LIN {X 0,Y 624.89,Z 336.382,A -85,B 0,C 180,E1 22685.786,E2 22685.786} C_VEL
LIN {X 0,Y 624.904,Z 336.388,A -85,B 0,C 180,E1 22682.935,E2 22682.935} C_VEL
LIN {X 0,Y 624.889,Z 336.39,A -85,B 0,C 180,E1 22679.725,E2 22679.725} C_VEL
LIN {X 0,Y 624.882,Z 336.387,A -85,B 0,C 180,E1 22676.973,E2 22676.973} C_VEL
LIN {X 0,Y 624.896,Z 336.39,A -85,B 0,C 180,E1 22673.753,E2 22673.753} C_VEL
LIN {X 0,Y 624.864,Z 336.382,A -85,B 0,C 180,E1 22671.071,E2 22671.071} C_VEL
LIN {X 0,Y 624.941,Z 336.367,A -85,B 0,C 180,E1 22668.089,E2 22668.089} C_VEL
LIN {X 0,Y 624.856,Z 336.372,A -85,B 0,C 180,E1 22665.129,E2 22665.129} C_VEL
LIN {X 0,Y 624.887,Z 336.388,A -85,B 0,C 180,E1 22662.397,E2 22662.397} C_VEL
LIN {X 0,Y 624.855,Z 336.37,A -85,B 0,C 180,E1 22659.192,E2 22659.192} C_VEL
LIN {X 0,Y 624.852,Z 336.393,A -85,B 0,C 180,E1 22656.618,E2 22656.618} C_VEL
LIN {X 0,Y 624.897,Z 336.367,A -85,B 0,C 180,E1 22653.485,E2 22653.485} C_VEL
LIN {X 0,Y 624.852,Z 336.389,A -85,B 0,C 180,E1 22650.681,E2 22650.681} C_VEL
LIN {X 0,Y 624.926,Z 336.387,A -85,B 0,C 180,E1 22647.805,E2 22647.805} C_VEL
LIN {X 0,Y 624.867,Z 336.396,A -85,B 0,C 180,E1 22644.826,E2 22644.826} C_VEL
LIN {X 0,Y 624.909,Z 336.51,A -85,B 0,C 180,E1 22644.021,E2 22644.021} C_VEL
LIN {X 0,Y 626.185,Z 339.775,A -85,B 0,C 180,E1 22643.558,E2 22643.558} C_VEL
LIN {X 0,Y 627.184,Z 341.437,A -85,B 0,C 180,E1 22643.284,E2 22643.284} C_VEL
LIN {X 0,Y 631.826,Z 350.571,A -85,B 0,C 180,E1 22641.946,E2 22641.946} C_VEL
LIN {X 0,Y 646.023,Z 370.4,A -85,B 0,C 180,E1 22640.049,E2 22640.049} C_VEL
LIN {X 0,Y 658.613,Z 388.736,A -85,B 0,C 180,E1 22638.466,E2 22638.466} C_VEL
LIN {X 0,Y 661.685,Z 393.59,A -85,B 0,C 180,E1 22638.09,E2 22638.09} C_VEL
LIN {X 0,Y 657.538,Z 599.762,A -85,B 0,C 180,E1 22635.27,E2 22635.27} C_VEL
LIN {X 0,Y 653.324,Z 821.102,A -85,B 0,C 180,E1 22632.317,E2 22632.317} C_VEL
LIN {X 0,Y 652.435,Z 844.522,A -85,B 0,C 180,E1 22631.931,E2 22631.931} C_VEL
LIN {X 0,Y 651.298,Z 867.206,A -85,B 0,C 180,E1 22631.437,E2 22631.437} C_VEL
LIN {X 0,Y 649.719,Z 893.305,A -85,B 0,C 180,E1 22630.717,E2 22630.717} C_VEL
LIN {X 0,Y 647.798,Z 918.713,A -85,B 0,C 180,E1 22629.833,E2 22629.833} C_VEL
LIN {X 0,Y 645.976,Z 940.579,A -85,B 0,C 180,E1 22628.935,E2 22628.935} C_VEL
LIN {X 0,Y 644.088,Z 961.696,A -85,B 0,C 180,E1 22627.934,E2 22627.934} C_VEL
LIN {X 0,Y 641.747,Z 986.505,A -85,B 0,C 180,E1 22626.581,E2 22626.581} C_VEL
LIN {X 0,Y 639.476,Z 1008.583,A -85,B 0,C 180,E1 22625.183,E2 22625.183} C_VEL
LIN {X 0,Y 637.567,Z 1026.895,A -85,B 0,C 180,E1 22623.885,E2 22623.885} C_VEL
LIN {X 0,Y 635.699,Z 1044.654,A -85,B 0,C 180,E1 22622.489,E2 22622.489} C_VEL
LIN {X 0,Y 633.544,Z 1065.5,A -85,B 0,C 180,E1 22620.667,E2 22620.667} C_VEL
LIN {X 0,Y 631.512,Z 1085.194,A -85,B 0,C 180,E1 22618.697,E2 22618.697} C_VEL
LIN {X 0,Y 630.037,Z 1100.529,A -85,B 0,C 180,E1 22616.994,E2 22616.994} C_VEL
LIN {X 0,Y 628.438,Z 1118.006,A -85,B 0,C 180,E1 22614.837,E2 22614.837} C_VEL
LIN {X 0,Y 627.119,Z 1133.826,A -85,B 0,C 180,E1 22612.597,E2 22612.597} C_VEL
LIN {X 0,Y 626.192,Z 1146.58,A -85,B 0,C 180,E1 22610.566,E2 22610.566} C_VEL
LIN {X 0,Y 625.357,Z 1159.888,A -85,B 0,C 180,E1 22608.167,E2 22608.167} C_VEL
LIN {X 0,Y 624.744,Z 1171.078,A -85,B 0,C 180,E1 22605.788,E2 22605.788} C_VEL
LIN {X 0,Y 624.417,Z 1179.159,A -85,B 0,C 180,E1 22603.804,E2 22603.804} C_VEL
LIN {X 0,Y 624.174,Z 1186.705,A -85,B 0,C 180,E1 22601.645,E2 22601.645} C_VEL
LIN {X 0,Y 624.015,Z 1193.594,A -85,B 0,C 180,E1 22599.221,E2 22599.221} C_VEL
LIN {X 0,Y 623.939,Z 1198.918,A -85,B 0,C 180,E1 22596.718,E2 22596.718} C_VEL
LIN {X 0,Y 623.915,Z 1202.24,A -85,B 0,C 180,E1 22594.504,E2 22594.504} C_VEL
LIN {X 0,Y 623.912,Z 1204.382,A -85,B 0,C 180,E1 22592.113,E2 22592.113} C_VEL
LIN {X 0,Y 623.892,Z 1204.894,A -85,B 0,C 180,E1 22589.541,E2 22589.541} C_VEL
LIN {X 0,Y 623.911,Z 1204.004,A -85,B 0,C 180,E1 22587.337,E2 22587.337} C_VEL
LIN {X 0,Y 623.923,Z 1201.672,A -85,B 0,C 180,E1 22585.036,E2 22585.036} C_VEL
LIN {X 0,Y 623.958,Z 1197.543,A -85,B 0,C 180,E1 22582.542,E2 22582.542} C_VEL
LIN {X 0,Y 624.046,Z 1191.873,A -85,B 0,C 180,E1 22580.129,E2 22580.129} C_VEL
LIN {X 0,Y 624.21,Z 1184.888,A -85,B 0,C 180,E1 22577.794,E2 22577.794} C_VEL
LIN {X 0,Y 624.578,Z 1175.442,A -85,B 0,C 180,E1 22575.229,E2 22575.229} C_VEL
LIN {X 0,Y 625.05,Z 1164.999,A -85,B 0,C 180,E1 22572.882,E2 22572.882} C_VEL
LIN {X 0,Y 625.664,Z 1154.466,A -85,B 0,C 180,E1 22570.821,E2 22570.821} C_VEL
LIN {X 0,Y 626.612,Z 1140.788,A -85,B 0,C 180,E1 22568.469,E2 22568.469} C_VEL
LIN {X 0,Y 627.822,Z 1125.095,A -85,B 0,C 180,E1 22566.139,E2 22566.139} C_VEL
LIN {X 0,Y 629.06,Z 1111.083,A -85,B 0,C 180,E1 22564.283,E2 22564.283} C_VEL
LIN {X 0,Y 630.77,Z 1092.862,A -85,B 0,C 180,E1 22562.12,E2 22562.12} C_VEL
LIN {X 0,Y 632.664,Z 1073.813,A -85,B 0,C 180,E1 22560.144,E2 22560.144} C_VEL
LIN {X 0,Y 634.359,Z 1057.391,A -85,B 0,C 180,E1 22558.606,E2 22558.606} C_VEL
LIN {X 0,Y 636.32,Z 1038.638,A -85,B 0,C 180,E1 22557.017,E2 22557.017} C_VEL
LIN {X 0,Y 638.858,Z 1014.535,A -85,B 0,C 180,E1 22555.222,E2 22555.222} C_VEL
LIN {X 0,Y 640.898,Z 994.594,A -85,B 0,C 180,E1 22553.916,E2 22553.916} C_VEL
LIN {X 0,Y 642.856,Z 974.946,A -85,B 0,C 180,E1 22552.769,E2 22552.769} C_VEL
LIN {X 0,Y 645.084,Z 951.666,A -85,B 0,C 180,E1 22551.571,E2 22551.571} C_VEL
LIN {X 0,Y 647.218,Z 926.44,A -85,B 0,C 180,E1 22550.47,E2 22550.47} C_VEL
LIN {X 0,Y 648.844,Z 904.861,A -85,B 0,C 180,E1 22549.668,E2 22549.668} C_VEL
LIN {X 0,Y 650.326,Z 883.219,A -85,B 0,C 180,E1 22548.988,E2 22548.988} C_VEL
LIN {X 0,Y 651.688,Z 860.13,A -85,B 0,C 180,E1 22548.394,E2 22548.394} C_VEL
LIN {X 0,Y 652.995,Z 831.823,A -85,B 0,C 180,E1 22547.842,E2 22547.842} C_VEL
LIN {X 0,Y 654.187,Z 777.579,A -85,B 0,C 180,E1 22547.102,E2 22547.102} C_VEL
LIN {X 0,Y 658.412,Z 555.546,A -85,B 0,C 180,E1 22544.133,E2 22544.133} C_VEL
LIN {X 0,Y 661.622,Z 393.144,A -85,B 0,C 180,E1 22541.897,E2 22541.897} C_VEL
LIN {X 0,Y 647.935,Z 373.153,A -85,B 0,C 180,E1 22540.199,E2 22540.199} C_VEL
LIN {X 0,Y 638.133,Z 359.287,A -85,B 0,C 180,E1 22538.898,E2 22538.898} C_VEL
LIN {X 0,Y 631.374,Z 349.693,A -85,B 0,C 180,E1 22537.913,E2 22537.913} C_VEL
LIN {X 0,Y 627.309,Z 341.424,A -85,B 0,C 180,E1 22536.594,E2 22536.594} C_VEL
LIN {X 0,Y 625.187,Z 337.75,A -85,B 0,C 180,E1 22535.942,E2 22535.942} C_VEL
LIN {X 0,Y 624.876,Z 336.385,A -85,B 0,C 180,E1 22535.736,E2 22535.736} C_VEL
LIN {X 0,Y 624.878,Z 336.391,A -85,B 0,C 180,E1 22532.96,E2 22532.96} C_VEL
LIN {X 0,Y 624.872,Z 336.375,A -85,B 0,C 180,E1 22529.633,E2 22529.633} C_VEL
LIN {X 0,Y 624.86,Z 336.37,A -85,B 0,C 180,E1 22526.966,E2 22526.966} C_VEL
LIN {X 0,Y 624.91,Z 336.391,A -85,B 0,C 180,E1 22523.88,E2 22523.88} C_VEL
LIN {X 0,Y 624.848,Z 336.368,A -85,B 0,C 180,E1 22521.103,E2 22521.103} C_VEL
LIN {X 0,Y 624.899,Z 336.383,A -85,B 0,C 180,E1 22518.277,E2 22518.277} C_VEL
LIN {X 0,Y 624.853,Z 336.384,A -85,B 0,C 180,E1 22515.215,E2 22515.215} C_VEL
LIN {X 0,Y 624.854,Z 336.38,A -85,B 0,C 180,E1 22512.57,E2 22512.57} C_VEL
LIN {X 0,Y 624.884,Z 336.388,A -85,B 0,C 180,E1 22509.393,E2 22509.393} C_VEL
LIN {X 0,Y 624.85,Z 336.372,A -85,B 0,C 180,E1 22506.708,E2 22506.708} C_VEL
LIN {X 0,Y 624.929,Z 336.381,A -85,B 0,C 180,E1 22503.761,E2 22503.761} C_VEL
LIN {X 0,Y 624.857,Z 336.362,A -85,B 0,C 180,E1 22500.733,E2 22500.733} C_VEL
LIN {X 0,Y 624.88,Z 336.388,A -85,B 0,C 180,E1 22498.074,E2 22498.074} C_VEL
LIN {X 0,Y 624.877,Z 336.356,A -85,B 0,C 180,E1 22494.859,E2 22494.859} C_VEL
LIN {X 0,Y 624.873,Z 336.392,A -85,B 0,C 180,E1 22492.183,E2 22492.183} C_VEL
LIN {X 0,Y 624.929,Z 336.355,A -85,B 0,C 180,E1 22489.117,E2 22489.117} C_VEL
LIN {X 0,Y 624.874,Z 336.39,A -85,B 0,C 180,E1 22486.206,E2 22486.206} C_VEL
LIN {X 0,Y 624.946,Z 336.36,A -85,B 0,C 180,E1 22483.262,E2 22483.262} C_VEL
LIN {X 0,Y 624.878,Z 336.366,A -85,B 0,C 180,E1 22480.196,E2 22480.196} C_VEL
LIN {X 0,Y 624.932,Z 336.391,A -85,B 0,C 180,E1 22477.319,E2 22477.319} C_VEL
LIN {X 0,Y 624.889,Z 336.375,A -85,B 0,C 180,E1 22474.2,E2 22474.2} C_VEL
LIN {X 0,Y 624.91,Z 336.39,A -85,B 0,C 180,E1 22471.418,E2 22471.418} C_VEL
LIN {X 0,Y 624.933,Z 336.553,A -85,B 0,C 180,E1 22469.363,E2 22469.363} C_VEL
LIN {X 0,Y 626.26,Z 339.858,A -85,B 0,C 180,E1 22468.844,E2 22468.844} C_VEL
LIN {X 0,Y 627.438,Z 341.862,A -85,B 0,C 180,E1 22468.499,E2 22468.499} C_VEL
LIN {X 0,Y 630.498,Z 346.011,A -85,B 0,C 180,E1 22468.043,E2 22468.043} C_VEL
LIN {X 0,Y 638.814,Z 357.205,A -85,B 0,C 180,E1 22466.862,E2 22466.862} C_VEL
LIN {X 0,Y 649.952,Z 372.837,A -85,B 0,C 180,E1 22465.398,E2 22465.398} C_VEL
LIN {X 0,Y 661.396,Z 389.816,A -85,B 0,C 180,E1 22463.978,E2 22463.978} C_VEL
LIN {X 0,Y 661.577,Z 391.519,A -85,B 0,C 180,E1 22463.934,E2 22463.934} C_VEL
LIN {X 0,Y 659.206,Z 504.502,A -85,B 0,C 180,E1 22462.383,E2 22462.383} C_VEL
LIN {X 0,Y 658.369,Z 512.206,A -85,B 0,C 180,E1 22462.34,E2 22462.34} C_VEL
LIN {X 0,Y 653.608,Z 532.876,A -85,B 0,C 180,E1 22462.456,E2 22462.456} C_VEL
LIN {X 0,Y 652.955,Z 539.485,A -85,B 0,C 180,E1 22462.413,E2 22462.413} C_VEL
LIN {X 0,Y 648.476,Z 760.283,A -85,B 0,C 180,E1 22459.432,E2 22459.432} C_VEL
LIN {X 0,Y 647.121,Z 819.424,A -85,B 0,C 180,E1 22458.626,E2 22458.626} C_VEL
LIN {X 0,Y 645.939,Z 846.309,A -85,B 0,C 180,E1 22458.126,E2 22458.126} C_VEL
LIN {X 0,Y 644.286,Z 872.533,A -85,B 0,C 180,E1 22457.46,E2 22457.46} C_VEL
LIN {X 0,Y 642.784,Z 893.338,A -85,B 0,C 180,E1 22456.807,E2 22456.807} C_VEL
LIN {X 0,Y 641.188,Z 912.912,A -85,B 0,C 180,E1 22456.091,E2 22456.091} C_VEL
LIN {X 0,Y 639.312,Z 933.875,A -85,B 0,C 180,E1 22455.203,E2 22455.203} C_VEL
LIN {X 0,Y 636.999,Z 958.427,A -85,B 0,C 180,E1 22453.999,E2 22453.999} C_VEL
LIN {X 0,Y 634.522,Z 981.775,A -85,B 0,C 180,E1 22452.655,E2 22452.655} C_VEL
LIN {X 0,Y 632.443,Z 1000.729,A -85,B 0,C 180,E1 22451.424,E2 22451.424} C_VEL
LIN {X 0,Y 630.472,Z 1018.453,A -85,B 0,C 180,E1 22450.144,E2 22450.144} C_VEL
LIN {X 0,Y 628.442,Z 1036.475,A -85,B 0,C 180,E1 22448.702,E2 22448.702} C_VEL
LIN {X 0,Y 625.996,Z 1058.337,A -85,B 0,C 180,E1 22446.737,E2 22446.737} C_VEL
LIN {X 0,Y 624.022,Z 1076.423,A -85,B 0,C 180,E1 22444.891,E2 22444.891} C_VEL
LIN {X 0,Y 622.369,Z 1092.43,A -85,B 0,C 180,E1 22443.075,E2 22443.075} C_VEL
LIN {X 0,Y 620.636,Z 1110.173,A -85,B 0,C 180,E1 22440.818,E2 22440.818} C_VEL
LIN {X 0,Y 619.314,Z 1125.112,A -85,B 0,C 180,E1 22438.652,E2 22438.652} C_VEL
LIN {X 0,Y 618.267,Z 1138.245,A -85,B 0,C 180,E1 22436.509,E2 22436.509} C_VEL
LIN {X 0,Y 617.357,Z 1151.707,A -85,B 0,C 180,E1 22433.986,E2 22433.986} C_VEL
LIN {X 0,Y 616.796,Z 1161.769,A -85,B 0,C 180,E1 22431.791,E2 22431.791} C_VEL
LIN {X 0,Y 616.438,Z 1169.628,A -85,B 0,C 180,E1 22429.815,E2 22429.815} C_VEL
LIN {X 0,Y 616.189,Z 1177.29,A -85,B 0,C 180,E1 22427.566,E2 22427.566} C_VEL
LIN {X 0,Y 616.012,Z 1184.218,A -85,B 0,C 180,E1 22425.03,E2 22425.03} C_VEL
LIN {X 0,Y 615.94,Z 1189.09,A -85,B 0,C 180,E1 22422.659,E2 22422.659} C_VEL
LIN {X 0,Y 615.918,Z 1192.403,A -85,B 0,C 180,E1 22420.381,E2 22420.381} C_VEL
LIN {X 0,Y 615.911,Z 1194.48,A -85,B 0,C 180,E1 22417.931,E2 22417.931} C_VEL
LIN {X 0,Y 615.897,Z 1194.873,A -85,B 0,C 180,E1 22415.403,E2 22415.403} C_VEL
LIN {X 0,Y 615.911,Z 1193.978,A -85,B 0,C 180,E1 22413.224,E2 22413.224} C_VEL
LIN {X 0,Y 615.922,Z 1191.675,A -85,B 0,C 180,E1 22410.93,E2 22410.93} C_VEL
LIN {X 0,Y 615.957,Z 1187.58,A -85,B 0,C 180,E1 22408.418,E2 22408.418} C_VEL
LIN {X 0,Y 616.059,Z 1181.985,A -85,B 0,C 180,E1 22405.998,E2 22405.998} C_VEL
LIN {X 0,Y 616.248,Z 1175.132,A -85,B 0,C 180,E1 22403.665,E2 22403.665} C_VEL
LIN {X 0,Y 616.611,Z 1166.051,A -85,B 0,C 180,E1 22401.138,E2 22401.138} C_VEL
LIN {X 0,Y 617.144,Z 1155.388,A -85,B 0,C 180,E1 22398.694,E2 22398.694} C_VEL
LIN {X 0,Y 617.824,Z 1144.736,A -85,B 0,C 180,E1 22396.573,E2 22396.573} C_VEL
LIN {X 0,Y 618.799,Z 1131.434,A -85,B 0,C 180,E1 22394.249,E2 22394.249} C_VEL
LIN {X 0,Y 620.121,Z 1115.714,A -85,B 0,C 180,E1 22391.869,E2 22391.869} C_VEL
LIN {X 0,Y 621.521,Z 1100.783,A -85,B 0,C 180,E1 22389.862,E2 22389.862} C_VEL
LIN {X 0,Y 623.428,Z 1082.331,A -85,B 0,C 180,E1 22387.659,E2 22387.659} C_VEL
LIN {X 0,Y 625.354,Z 1064.042,A -85,B 0,C 180,E1 22385.737,E2 22385.737} C_VEL
LIN {X 0,Y 627.208,Z 1047.276,A -85,B 0,C 180,E1 22384.15,E2 22384.15} C_VEL
LIN {X 0,Y 629.591,Z 1026.399,A -85,B 0,C 180,E1 22382.371,E2 22382.371} C_VEL
LIN {X 0,Y 632.056,Z 1004.368,A -85,B 0,C 180,E1 22380.737,E2 22380.737} C_VEL
LIN {X 0,Y 634.113,Z 985.502,A -85,B 0,C 180,E1 22379.487,E2 22379.487} C_VEL
LIN {X 0,Y 636.091,Z 966.892,A -85,B 0,C 180,E1 22378.383,E2 22378.383} C_VEL
LIN {X 0,Y 638.112,Z 946.922,A -85,B 0,C 180,E1 22377.329,E2 22377.329} C_VEL
LIN {X 0,Y 640.507,Z 921.876,A -85,B 0,C 180,E1 22376.179,E2 22376.179} C_VEL
LIN {X 0,Y 642.488,Z 897.06,A -85,B 0,C 180,E1 22375.229,E2 22375.229} C_VEL
LIN {X 0,Y 644.102,Z 875.213,A -85,B 0,C 180,E1 22374.529,E2 22374.529} C_VEL
LIN {X 0,Y 645.505,Z 852.967,A -85,B 0,C 180,E1 22373.941,E2 22373.941} C_VEL
LIN {X 0,Y 646.909,Z 825.987,A -85,B 0,C 180,E1 22373.386,E2 22373.386} C_VEL
LIN {X 0,Y 647.949,Z 787.5,A -85,B 0,C 180,E1 22372.84,E2 22372.84} C_VEL
LIN {X 0,Y 652.501,Z 561.879,A -85,B 0,C 180,E1 22369.805,E2 22369.805} C_VEL
LIN {X 0,Y 656.11,Z 393.795,A -85,B 0,C 180,E1 22367.479,E2 22367.479} C_VEL
LIN {X 0,Y 643.7,Z 375.505,A -85,B 0,C 180,E1 22365.902,E2 22365.902} C_VEL
LIN {X 0,Y 631.034,Z 357.881,A -85,B 0,C 180,E1 22364.202,E2 22364.202} C_VEL
LIN {X 0,Y 623.545,Z 347.824,A -85,B 0,C 180,E1 22363.167,E2 22363.167} C_VEL
LIN {X 0,Y 619.861,Z 343.139,A -85,B 0,C 180,E1 22362.649,E2 22362.649} C_VEL
LIN {X 0,Y 618.834,Z 341.576,A -85,B 0,C 180,E1 22362.485,E2 22362.485} C_VEL
LIN {X 0,Y 617.176,Z 338.348,A -85,B 0,C 180,E1 22361.959,E2 22361.959} C_VEL
LIN {X 0,Y 617.004,Z 337.37,A -85,B 0,C 180,E1 22361.802,E2 22361.802} C_VEL
LIN {X 0,Y 616.995,Z 337.378,A -85,B 0,C 180,E1 22358.603,E2 22358.603} C_VEL
LIN {X 0,Y 617.013,Z 337.368,A -85,B 0,C 180,E1 22355.401,E2 22355.401} C_VEL
LIN {X 0,Y 616.977,Z 337.38,A -85,B 0,C 180,E1 22352.221,E2 22352.221} C_VEL
LIN {X 0,Y 617.018,Z 337.374,A -85,B 0,C 180,E1 22349.088,E2 22349.088} C_VEL
LIN {X 0,Y 616.964,Z 337.339,A -85,B 0,C 180,E1 22345.95,E2 22345.95} C_VEL
LIN {X 0,Y 617.017,Z 337.373,A -85,B 0,C 180,E1 22342.888,E2 22342.888} C_VEL
LIN {X 0,Y 616.956,Z 337.338,A -85,B 0,C 180,E1 22339.799,E2 22339.799} C_VEL
LIN {X 0,Y 617.018,Z 337.374,A -85,B 0,C 180,E1 22336.668,E2 22336.668} C_VEL
LIN {X 0,Y 616.949,Z 337.33,A -85,B 0,C 180,E1 22333.687,E2 22333.687} C_VEL
LIN {X 0,Y 617.015,Z 337.371,A -85,B 0,C 180,E1 22330.646,E2 22330.646} C_VEL
LIN {X 0,Y 616.948,Z 337.378,A -85,B 0,C 180,E1 22327.637,E2 22327.637} C_VEL
LIN {X 0,Y 617.003,Z 337.363,A -85,B 0,C 180,E1 22324.648,E2 22324.648} C_VEL
LIN {X 0,Y 616.942,Z 337.369,A -85,B 0,C 180,E1 22321.579,E2 22321.579} C_VEL
LIN {X 0,Y 616.965,Z 337.376,A -85,B 0,C 180,E1 22318.793,E2 22318.793} C_VEL
LIN {X 0,Y 616.945,Z 337.375,A -85,B 0,C 180,E1 22315.631,E2 22315.631} C_VEL
LIN {X 0,Y 616.943,Z 337.379,A -85,B 0,C 180,E1 22312.831,E2 22312.831} C_VEL
LIN {X 0,Y 616.941,Z 337.381,A -85,B 0,C 180,E1 22309.542,E2 22309.542} C_VEL
LIN {X 0,Y 616.923,Z 337.342,A -85,B 0,C 180,E1 22306.789,E2 22306.789} C_VEL
LIN {X 0,Y 616.955,Z 337.383,A -85,B 0,C 180,E1 22303.62,E2 22303.62} C_VEL
LIN {X 0,Y 616.912,Z 337.346,A -85,B 0,C 180,E1 22300.79,E2 22300.79} C_VEL
LIN {X 0,Y 616.977,Z 337.38,A -85,B 0,C 180,E1 22297.714,E2 22297.714} C_VEL
LIN {X 0,Y 616.905,Z 337.342,A -85,B 0,C 180,E1 22294.744,E2 22294.744} C_VEL
LIN {X 0,Y 616.993,Z 337.371,A -85,B 0,C 180,E1 22291.651,E2 22291.651} C_VEL
LIN {X 0,Y 616.917,Z 337.375,A -85,B 0,C 180,E1 22288.758,E2 22288.758} C_VEL
LIN {X 0,Y 616.972,Z 337.38,A -85,B 0,C 180,E1 22285.893,E2 22285.893} C_VEL
LIN {X 0,Y 616.956,Z 337.573,A -85,B 0,C 180,E1 22284.876,E2 22284.876} C_VEL
LIN {X 0,Y 618.245,Z 340.888,A -85,B 0,C 180,E1 22284.392,E2 22284.392} C_VEL
LIN {X 0,Y 619.281,Z 342.41,A -85,B 0,C 180,E1 22284.119,E2 22284.119} C_VEL
LIN {X 0,Y 623.249,Z 350.434,A -85,B 0,C 180,E1 22282.927,E2 22282.927} C_VEL
LIN {X 0,Y 633.22,Z 364.022,A -85,B 0,C 180,E1 22281.553,E2 22281.553} C_VEL
LIN {X 0,Y 642.371,Z 376.825,A -85,B 0,C 180,E1 22280.328,E2 22280.328} C_VEL
LIN {X 0,Y 654.513,Z 394.616,A -85,B 0,C 180,E1 22278.776,E2 22278.776} C_VEL
LIN {X 0,Y 656.246,Z 397.425,A -85,B 0,C 180,E1 22278.558,E2 22278.558} C_VEL
LIN {X 0,Y 651.843,Z 602.744,A -85,B 0,C 180,E1 22275.731,E2 22275.731} C_VEL
LIN {X 0,Y 647.363,Z 822.354,A -85,B 0,C 180,E1 22272.777,E2 22272.777} C_VEL
LIN {X 0,Y 646.445,Z 844.984,A -85,B 0,C 180,E1 22272.398,E2 22272.398} C_VEL
LIN {X 0,Y 645.253,Z 867.36,A -85,B 0,C 180,E1 22271.907,E2 22271.907} C_VEL
LIN {X 0,Y 643.578,Z 893.513,A -85,B 0,C 180,E1 22271.182,E2 22271.182} C_VEL
LIN {X 0,Y 641.557,Z 918.71,A -85,B 0,C 180,E1 22270.3,E2 22270.3} C_VEL
LIN {X 0,Y 639.625,Z 940.576,A -85,B 0,C 180,E1 22269.396,E2 22269.396} C_VEL
LIN {X 0,Y 637.616,Z 961.692,A -85,B 0,C 180,E1 22268.388,E2 22268.388} C_VEL
LIN {X 0,Y 635.13,Z 986.242,A -85,B 0,C 180,E1 22267.043,E2 22267.043} C_VEL
LIN {X 0,Y 632.685,Z 1008.58,A -85,B 0,C 180,E1 22265.617,E2 22265.617} C_VEL
LIN {X 0,Y 630.637,Z 1026.953,A -85,B 0,C 180,E1 22264.304,E2 22264.304} C_VEL
LIN {X 0,Y 628.618,Z 1044.939,A -85,B 0,C 180,E1 22262.876,E2 22262.876} C_VEL
LIN {X 0,Y 626.329,Z 1065.681,A -85,B 0,C 180,E1 22261.04,E2 22261.04} C_VEL
LIN {X 0,Y 624.16,Z 1084.985,A -85,B 0,C 180,E1 22259.091,E2 22259.091} C_VEL
LIN {X 0,Y 622.551,Z 1100.527,A -85,B 0,C 180,E1 22257.345,E2 22257.345} C_VEL
LIN {X 0,Y 620.834,Z 1118.04,A -85,B 0,C 180,E1 22255.158,E2 22255.158} C_VEL
LIN {X 0,Y 619.411,Z 1133.828,A -85,B 0,C 180,E1 22252.895,E2 22252.895} C_VEL
LIN {X 0,Y 618.402,Z 1146.578,A -85,B 0,C 180,E1 22250.837,E2 22250.837} C_VEL
LIN {X 0,Y 617.489,Z 1159.947,A -85,B 0,C 180,E1 22248.395,E2 22248.395} C_VEL
LIN {X 0,Y 616.834,Z 1171.079,A -85,B 0,C 180,E1 22245.996,E2 22245.996} C_VEL
LIN {X 0,Y 616.462,Z 1179.16,A -85,B 0,C 180,E1 22243.986,E2 22243.986} C_VEL
LIN {X 0,Y 616.199,Z 1186.399,A -85,B 0,C 180,E1 22241.893,E2 22241.893} C_VEL
LIN {X 0,Y 616.034,Z 1193.351,A -85,B 0,C 180,E1 22239.436,E2 22239.436} C_VEL
LIN {X 0,Y 615.943,Z 1198.756,A -85,B 0,C 180,E1 22236.9,E2 22236.9} C_VEL
LIN {X 0,Y 615.914,Z 1202.2,A -85,B 0,C 180,E1 22234.593,E2 22234.593} C_VEL
LIN {X 0,Y 615.911,Z 1204.326,A -85,B 0,C 180,E1 22232.233,E2 22232.233} C_VEL
LIN {X 0,Y 615.894,Z 1204.917,A -85,B 0,C 180,E1 22229.628,E2 22229.628} C_VEL
LIN {X 0,Y 615.912,Z 1204.001,A -85,B 0,C 180,E1 22227.302,E2 22227.302} C_VEL
LIN {X 0,Y 615.925,Z 1201.669,A -85,B 0,C 180,E1 22224.971,E2 22224.971} C_VEL
LIN {X 0,Y 615.96,Z 1197.543,A -85,B 0,C 180,E1 22222.445,E2 22222.445} C_VEL
LIN {X 0,Y 616.061,Z 1191.87,A -85,B 0,C 180,E1 22220,E2 22220} C_VEL
LIN {X 0,Y 616.231,Z 1185.188,A -85,B 0,C 180,E1 22217.728,E2 22217.728} C_VEL
LIN {X 0,Y 616.603,Z 1176.301,A -85,B 0,C 180,E1 22215.251,E2 22215.251} C_VEL
LIN {X 0,Y 617.135,Z 1165.456,A -85,B 0,C 180,E1 22212.753,E2 22212.753} C_VEL
LIN {X 0,Y 617.794,Z 1154.969,A -85,B 0,C 180,E1 22210.662,E2 22210.662} C_VEL
LIN {X 0,Y 618.707,Z 1142.536,A -85,B 0,C 180,E1 22208.479,E2 22208.479} C_VEL
LIN {X 0,Y 620.047,Z 1126.494,A -85,B 0,C 180,E1 22206.023,E2 22206.023} C_VEL
LIN {X 0,Y 621.426,Z 1111.851,A -85,B 0,C 180,E1 22204.047,E2 22204.047} C_VEL
LIN {X 0,Y 623.059,Z 1095.439,A -85,B 0,C 180,E1 22202.057,E2 22202.057} C_VEL
LIN {X 0,Y 625.237,Z 1075.258,A -85,B 0,C 180,E1 22199.904,E2 22199.904} C_VEL
LIN {X 0,Y 627.086,Z 1058.5,A -85,B 0,C 180,E1 22198.307,E2 22198.307} C_VEL
LIN {X 0,Y 629.039,Z 1041.009,A -85,B 0,C 180,E1 22196.799,E2 22196.799} C_VEL
LIN {X 0,Y 631.556,Z 1018.933,A -85,B 0,C 180,E1 22195.096,E2 22195.096} C_VEL
LIN {X 0,Y 634.035,Z 996.245,A -85,B 0,C 180,E1 22193.577,E2 22193.577} C_VEL
LIN {X 0,Y 636.012,Z 977.642,A -85,B 0,C 180,E1 22192.47,E2 22192.47} C_VEL
LIN {X 0,Y 638.03,Z 957.693,A -85,B 0,C 180,E1 22191.412,E2 22191.412} C_VEL
LIN {X 0,Y 640.078,Z 936.074,A -85,B 0,C 180,E1 22190.407,E2 22190.407} C_VEL
LIN {X 0,Y 642.392,Z 908.556,A -85,B 0,C 180,E1 22189.325,E2 22189.325} C_VEL
LIN {X 0,Y 644.095,Z 885.246,A -85,B 0,C 180,E1 22188.574,E2 22188.574} C_VEL
LIN {X 0,Y 645.475,Z 863.37,A -85,B 0,C 180,E1 22187.996,E2 22187.996} C_VEL
LIN {X 0,Y 646.72,Z 839.343,A -85,B 0,C 180,E1 22187.494,E2 22187.494} C_VEL
LIN {X 0,Y 647.825,Z 803.917,A -85,B 0,C 180,E1 22186.97,E2 22186.97} C_VEL
LIN {X 0,Y 652.326,Z 579.686,A -85,B 0,C 180,E1 22183.957,E2 22183.957} C_VEL
LIN {X 0,Y 656.24,Z 397.189,A -85,B 0,C 180,E1 22181.438,E2 22181.438} C_VEL
LIN {X 0,Y 643.845,Z 378.971,A -85,B 0,C 180,E1 22179.867,E2 22179.867} C_VEL
LIN {X 0,Y 634.433,Z 365.48,A -85,B 0,C 180,E1 22178.584,E2 22178.584} C_VEL
LIN {X 0,Y 627.281,Z 355.576,A -85,B 0,C 180,E1 22177.54,E2 22177.54} C_VEL
LIN {X 0,Y 622.645,Z 349.332,A -85,B 0,C 180,E1 22176.798,E2 22176.798} C_VEL
LIN {X 0,Y 621.318,Z 346.29,A -85,B 0,C 180,E1 22176.315,E2 22176.315} C_VEL
LIN {X 0,Y 619.384,Z 342.337,A -85,B 0,C 180,E1 22175.646,E2 22175.646} C_VEL
LIN {X 0,Y 617.282,Z 338.887,A -85,B 0,C 180,E1 22174.989,E2 22174.989} C_VEL
LIN {X 0,Y 616.966,Z 337.376,A -85,B 0,C 180,E1 22174.749,E2 22174.749} C_VEL
LIN {X 0,Y 616.929,Z 337.363,A -85,B 0,C 180,E1 22171.568,E2 22171.568} C_VEL
LIN {X 0,Y 616.929,Z 337.379,A -85,B 0,C 180,E1 22168.933,E2 22168.933} C_VEL
LIN {X 0,Y 616.946,Z 337.352,A -85,B 0,C 180,E1 22165.744,E2 22165.744} C_VEL
LIN {X 0,Y 616.915,Z 337.373,A -85,B 0,C 180,E1 22162.988,E2 22162.988} C_VEL
LIN {X 0,Y 616.989,Z 337.365,A -85,B 0,C 180,E1 22159.961,E2 22159.961} C_VEL
LIN {X 0,Y 616.905,Z 337.351,A -85,B 0,C 180,E1 22156.963,E2 22156.963} C_VEL
LIN {X 0,Y 616.991,Z 337.379,A -85,B 0,C 180,E1 22153.973,E2 22153.973} C_VEL
LIN {X 0,Y 616.907,Z 337.35,A -85,B 0,C 180,E1 22150.932,E2 22150.932} C_VEL
LIN {X 0,Y 616.952,Z 337.382,A -85,B 0,C 180,E1 22148.106,E2 22148.106} C_VEL
LIN {X 0,Y 616.919,Z 337.358,A -85,B 0,C 180,E1 22144.928,E2 22144.928} C_VEL
LIN {X 0,Y 616.941,Z 337.376,A -85,B 0,C 180,E1 22142.136,E2 22142.136} C_VEL
LIN {X 0,Y 616.932,Z 337.367,A -85,B 0,C 180,E1 22138.886,E2 22138.886} C_VEL
LIN {X 0,Y 616.93,Z 337.368,A -85,B 0,C 180,E1 22136.19,E2 22136.19} C_VEL
LIN {X 0,Y 616.965,Z 337.37,A -85,B 0,C 180,E1 22133.018,E2 22133.018} C_VEL
LIN {X 0,Y 616.93,Z 337.355,A -85,B 0,C 180,E1 22130.195,E2 22130.195} C_VEL
LIN {X 0,Y 616.998,Z 337.377,A -85,B 0,C 180,E1 22127.077,E2 22127.077} C_VEL
LIN {X 0,Y 616.932,Z 337.343,A -85,B 0,C 180,E1 22124.2,E2 22124.2} C_VEL
LIN {X 0,Y 617.013,Z 337.361,A -85,B 0,C 180,E1 22121.15,E2 22121.15} C_VEL
LIN {X 0,Y 616.942,Z 337.375,A -85,B 0,C 180,E1 22118.114,E2 22118.114} C_VEL
LIN {X 0,Y 617.003,Z 337.343,A -85,B 0,C 180,E1 22115.161,E2 22115.161} C_VEL
LIN {X 0,Y 616.949,Z 337.375,A -85,B 0,C 180,E1 22112.038,E2 22112.038} C_VEL
LIN {X 0,Y 616.983,Z 337.474,A -85,B 0,C 180,E1 22110.348,E2 22110.348} C_VEL
LIN {X 0,Y 618.254,Z 340.857,A -85,B 0,C 180,E1 22109.803,E2 22109.803} C_VEL
LIN {X 0,Y 619.653,Z 342.616,A -85,B 0,C 180,E1 22109.49,E2 22109.49} C_VEL
LIN {X 0,Y 622.74,Z 346.839,A -85,B 0,C 180,E1 22109.002,E2 22109.002} C_VEL
LIN {X 0,Y 624.47,Z 349.091,A -85,B 0,C 180,E1 22108.736,E2 22108.736} C_VEL
LIN {X 0,Y 633.333,Z 360.888,A -85,B 0,C 180,E1 22107.428,E2 22107.428} C_VEL
LIN {X 0,Y 645.586,Z 378.208,A -85,B 0,C 180,E1 22105.764,E2 22105.764} C_VEL
LIN {X 0,Y 656.173,Z 394,A -85,B 0,C 180,E1 22104.422,E2 22104.422} C_VEL
LIN {X 0,Y 652.955,Z 539.485,A -85,B 0,C 180,E1 22102.413,E2 22102.413} C_VEL
LIN {X 0,Y 652.115,Z 547.19,A -85,B 0,C 180,E1 22102.37,E2 22102.37} C_VEL
LIN {X 0,Y 647.354,Z 567.86,A -85,B 0,C 180,E1 22102.488,E2 22102.488} C_VEL
LIN {X 0,Y 646.685,Z 574.472,A -85,B 0,C 180,E1 22102.446,E2 22102.446} C_VEL
LIN {X 0,Y 641.838,Z 800.695,A -85,B 0,C 180,E1 22099.384,E2 22099.384} C_VEL
LIN {X 0,Y 640.673,Z 832.128,A -85,B 0,C 180,E1 22098.894,E2 22098.894} C_VEL
LIN {X 0,Y 639.39,Z 855.107,A -85,B 0,C 180,E1 22098.401,E2 22098.401} C_VEL
LIN {X 0,Y 637.929,Z 876.741,A -85,B 0,C 180,E1 22097.818,E2 22097.818} C_VEL
LIN {X 0,Y 636.071,Z 900.688,A -85,B 0,C 180,E1 22097.032,E2 22097.032} C_VEL
LIN {X 0,Y 633.64,Z 927.601,A -85,B 0,C 180,E1 22095.953,E2 22095.953} C_VEL
LIN {X 0,Y 631.556,Z 948.323,A -85,B 0,C 180,E1 22094.976,E2 22094.976} C_VEL
LIN {X 0,Y 629.504,Z 967.412,A -85,B 0,C 180,E1 22093.956,E2 22093.956} C_VEL
LIN {X 0,Y 627.378,Z 986.216,A -85,B 0,C 180,E1 22092.828,E2 22092.828} C_VEL
LIN {X 0,Y 625.133,Z 1005.507,A -85,B 0,C 180,E1 22091.534,E2 22091.534} C_VEL
LIN {X 0,Y 622.208,Z 1029.643,A -85,B 0,C 180,E1 22089.694,E2 22089.694} C_VEL
LIN {X 0,Y 619.991,Z 1048.117,A -85,B 0,C 180,E1 22088.092,E2 22088.092} C_VEL
LIN {X 0,Y 618.023,Z 1064.906,A -85,B 0,C 180,E1 22086.477,E2 22086.477} C_VEL
LIN {X 0,Y 615.824,Z 1084.254,A -85,B 0,C 180,E1 22084.404,E2 22084.404} C_VEL
LIN {X 0,Y 613.91,Z 1101.564,A -85,B 0,C 180,E1 22082.29,E2 22082.29} C_VEL
LIN {X 0,Y 612.416,Z 1116.385,A -85,B 0,C 180,E1 22080.265,E2 22080.265} C_VEL
LIN {X 0,Y 610.972,Z 1132.32,A -85,B 0,C 180,E1 22077.801,E2 22077.801} C_VEL
LIN {X 0,Y 609.963,Z 1145.041,A -85,B 0,C 180,E1 22075.538,E2 22075.538} C_VEL
LIN {X 0,Y 609.236,Z 1155.603,A -85,B 0,C 180,E1 22073.401,E2 22073.401} C_VEL
LIN {X 0,Y 608.644,Z 1166.738,A -85,B 0,C 180,E1 22070.783,E2 22070.783} C_VEL
LIN {X 0,Y 608.262,Z 1175.164,A -85,B 0,C 180,E1 22068.397,E2 22068.397} C_VEL
LIN {X 0,Y 608.085,Z 1181.744,A -85,B 0,C 180,E1 22066.134,E2 22066.134} C_VEL
LIN {X 0,Y 607.967,Z 1187.558,A -85,B 0,C 180,E1 22063.602,E2 22063.602} C_VEL
LIN {X 0,Y 607.924,Z 1191.614,A -85,B 0,C 180,E1 22061.094,E2 22061.094} C_VEL
LIN {X 0,Y 607.914,Z 1193.919,A -85,B 0,C 180,E1 22058.798,E2 22058.798} C_VEL
LIN {X 0,Y 607.891,Z 1194.85,A -85,B 0,C 180,E1 22056.611,E2 22056.611} C_VEL
LIN {X 0,Y 607.915,Z 1194.598,A -85,B 0,C 180,E1 22054.244,E2 22054.244} C_VEL
LIN {X 0,Y 607.919,Z 1192.671,A -85,B 0,C 180,E1 22051.696,E2 22051.696} C_VEL
LIN {X 0,Y 607.942,Z 1189.386,A -85,B 0,C 180,E1 22049.34,E2 22049.34} C_VEL
LIN {X 0,Y 608.015,Z 1184.732,A -85,B 0,C 180,E1 22046.983,E2 22046.983} C_VEL
LIN {X 0,Y 608.198,Z 1177.747,A -85,B 0,C 180,E1 22044.339,E2 22044.339} C_VEL
LIN {X 0,Y 608.457,Z 1170.194,A -85,B 0,C 180,E1 22042.065,E2 22042.065} C_VEL
LIN {X 0,Y 608.875,Z 1162.049,A -85,B 0,C 180,E1 22039.975,E2 22039.975} C_VEL
LIN {X 0,Y 609.472,Z 1152.171,A -85,B 0,C 180,E1 22037.782,E2 22037.782} C_VEL
LIN {X 0,Y 610.453,Z 1138.639,A -85,B 0,C 180,E1 22035.196,E2 22035.196} C_VEL
LIN {X 0,Y 611.552,Z 1125.619,A -85,B 0,C 180,E1 22033.035,E2 22033.035} C_VEL
LIN {X 0,Y 612.874,Z 1111.554,A -85,B 0,C 180,E1 22030.956,E2 22030.956} C_VEL
LIN {X 0,Y 614.769,Z 1093.734,A -85,B 0,C 180,E1 22028.634,E2 22028.634} C_VEL
LIN {X 0,Y 616.6,Z 1076.896,A -85,B 0,C 180,E1 22026.692,E2 22026.692} C_VEL
LIN {X 0,Y 618.646,Z 1059.55,A -85,B 0,C 180,E1 22024.896,E2 22024.896} C_VEL
LIN {X 0,Y 621.317,Z 1037.386,A -85,B 0,C 180,E1 22022.867,E2 22022.867} C_VEL
LIN {X 0,Y 623.546,Z 1018.662,A -85,B 0,C 180,E1 22021.35,E2 22021.35} C_VEL
LIN {X 0,Y 625.742,Z 1000.207,A -85,B 0,C 180,E1 22020.006,E2 22020.006} C_VEL
LIN {X 0,Y 628.197,Z 979.129,A -85,B 0,C 180,E1 22018.636,E2 22018.636} C_VEL
LIN {X 0,Y 630.911,Z 954.254,A -85,B 0,C 180,E1 22017.233,E2 22017.233} C_VEL
LIN {X 0,Y 633.021,Z 933.498,A -85,B 0,C 180,E1 22016.22,E2 22016.22} C_VEL
LIN {X 0,Y 635,Z 912.519,A -85,B 0,C 180,E1 22015.328,E2 22015.328} C_VEL
LIN {X 0,Y 636.789,Z 891.613,A -85,B 0,C 180,E1 22014.564,E2 22014.564} C_VEL
LIN {X 0,Y 638.791,Z 865.426,A -85,B 0,C 180,E1 22013.766,E2 22013.766} C_VEL
LIN {X 0,Y 640.32,Z 838.967,A -85,B 0,C 180,E1 22013.15,E2 22013.15} C_VEL
LIN {X 0,Y 641.33,Z 816.668,A -85,B 0,C 180,E1 22012.756,E2 22012.756} C_VEL
LIN {X 0,Y 645.82,Z 613.37,A -85,B 0,C 180,E1 22009.997,E2 22009.997} C_VEL
LIN {X 0,Y 650.748,Z 397.796,A -85,B 0,C 180,E1 22007.008,E2 22007.008} C_VEL
LIN {X 0,Y 639.624,Z 381.294,A -85,B 0,C 180,E1 22005.563,E2 22005.563} C_VEL
LIN {X 0,Y 627.324,Z 364.162,A -85,B 0,C 180,E1 22003.896,E2 22003.896} C_VEL
LIN {X 0,Y 618.536,Z 352.65,A -85,B 0,C 180,E1 22002.667,E2 22002.667} C_VEL
LIN {X 0,Y 614.915,Z 347.771,A -85,B 0,C 180,E1 22002.143,E2 22002.143} C_VEL
LIN {X 0,Y 611.866,Z 343.594,A -85,B 0,C 180,E1 22001.691,E2 22001.691} C_VEL
LIN {X 0,Y 610.293,Z 341.709,A -85,B 0,C 180,E1 22001.446,E2 22001.446} C_VEL
LIN {X 0,Y 609.077,Z 338.362,A -85,B 0,C 180,E1 22000.921,E2 22000.921} C_VEL
LIN {X 0,Y 609.062,Z 338.358,A -85,B 0,C 180,E1 21997.694,E2 21997.694} C_VEL
LIN {X 0,Y 609.045,Z 338.369,A -85,B 0,C 180,E1 21994.386,E2 21994.386} C_VEL
LIN {X 0,Y 609.078,Z 338.359,A -85,B 0,C 180,E1 21991.208,E2 21991.208} C_VEL
LIN {X 0,Y 609.032,Z 338.353,A -85,B 0,C 180,E1 21988.112,E2 21988.112} C_VEL
LIN {X 0,Y 609.074,Z 338.339,A -85,B 0,C 180,E1 21984.955,E2 21984.955} C_VEL
LIN {X 0,Y 609.022,Z 338.349,A -85,B 0,C 180,E1 21981.882,E2 21981.882} C_VEL
LIN {X 0,Y 609.077,Z 338.336,A -85,B 0,C 180,E1 21978.77,E2 21978.77} C_VEL
LIN {X 0,Y 609.017,Z 338.355,A -85,B 0,C 180,E1 21975.718,E2 21975.718} C_VEL
LIN {X 0,Y 609.074,Z 338.322,A -85,B 0,C 180,E1 21972.612,E2 21972.612} C_VEL
LIN {X 0,Y 609.011,Z 338.363,A -85,B 0,C 180,E1 21969.545,E2 21969.545} C_VEL
LIN {X 0,Y 609.077,Z 338.362,A -85,B 0,C 180,E1 21966.409,E2 21966.409} C_VEL
LIN {X 0,Y 609.003,Z 338.368,A -85,B 0,C 180,E1 21963.389,E2 21963.389} C_VEL
LIN {X 0,Y 609.077,Z 338.36,A -85,B 0,C 180,E1 21960.282,E2 21960.282} C_VEL
LIN {X 0,Y 608.996,Z 338.366,A -85,B 0,C 180,E1 21957.271,E2 21957.271} C_VEL
LIN {X 0,Y 609.067,Z 338.354,A -85,B 0,C 180,E1 21954.158,E2 21954.158} C_VEL
LIN {X 0,Y 608.986,Z 338.359,A -85,B 0,C 180,E1 21951.217,E2 21951.217} C_VEL
LIN {X 0,Y 609.049,Z 338.348,A -85,B 0,C 180,E1 21948.254,E2 21948.254} C_VEL
LIN {X 0,Y 608.98,Z 338.343,A -85,B 0,C 180,E1 21945.159,E2 21945.159} C_VEL
LIN {X 0,Y 609.017,Z 338.359,A -85,B 0,C 180,E1 21942.318,E2 21942.318} C_VEL
LIN {X 0,Y 608.974,Z 338.345,A -85,B 0,C 180,E1 21939.127,E2 21939.127} C_VEL
LIN {X 0,Y 608.981,Z 338.36,A -85,B 0,C 180,E1 21936.485,E2 21936.485} C_VEL
LIN {X 0,Y 608.986,Z 338.355,A -85,B 0,C 180,E1 21933.159,E2 21933.159} C_VEL
LIN {X 0,Y 608.987,Z 338.368,A -85,B 0,C 180,E1 21930.382,E2 21930.382} C_VEL
LIN {X 0,Y 609.001,Z 338.372,A -85,B 0,C 180,E1 21927.081,E2 21927.081} C_VEL
LIN {X 0,Y 609.05,Z 338.383,A -85,B 0,C 180,E1 21925.786,E2 21925.786} C_VEL
LIN {X 0,Y 610.42,Z 341.984,A -85,B 0,C 180,E1 21925.247,E2 21925.247} C_VEL
LIN {X 0,Y 611.375,Z 343.587,A -85,B 0,C 180,E1 21924.966,E2 21924.966} C_VEL
LIN {X 0,Y 613.148,Z 347.134,A -85,B 0,C 180,E1 21924.396,E2 21924.396} C_VEL
LIN {X 0,Y 614.785,Z 350.358,A -85,B 0,C 180,E1 21923.931,E2 21923.931} C_VEL
LIN {X 0,Y 628.629,Z 368.967,A -85,B 0,C 180,E1 21921.978,E2 21921.978} C_VEL
LIN {X 0,Y 639.151,Z 383.876,A -85,B 0,C 180,E1 21920.554,E2 21920.554} C_VEL
LIN {X 0,Y 650.504,Z 400.609,A -85,B 0,C 180,E1 21919.08,E2 21919.08} C_VEL
LIN {X 0,Y 650.839,Z 401.751,A -85,B 0,C 180,E1 21919.028,E2 21919.028} C_VEL
LIN {X 0,Y 646.174,Z 606.094,A -85,B 0,C 180,E1 21916.194,E2 21916.194} C_VEL
LIN {X 0,Y 641.467,Z 822.964,A -85,B 0,C 180,E1 21913.254,E2 21913.254} C_VEL
LIN {X 0,Y 640.514,Z 845.121,A -85,B 0,C 180,E1 21912.881,E2 21912.881} C_VEL
LIN {X 0,Y 639.273,Z 867.129,A -85,B 0,C 180,E1 21912.396,E2 21912.396} C_VEL
LIN {X 0,Y 637.531,Z 892.998,A -85,B 0,C 180,E1 21911.678,E2 21911.678} C_VEL
LIN {X 0,Y 635.362,Z 918.707,A -85,B 0,C 180,E1 21910.775,E2 21910.775} C_VEL
LIN {X 0,Y 633.39,Z 939.907,A -85,B 0,C 180,E1 21909.895,E2 21909.895} C_VEL
LIN {X 0,Y 631.299,Z 960.684,A -85,B 0,C 180,E1 21908.902,E2 21908.902} C_VEL
LIN {X 0,Y 628.881,Z 983.106,A -85,B 0,C 180,E1 21907.68,E2 21907.68} C_VEL
LIN {X 0,Y 626.013,Z 1007.843,A -85,B 0,C 180,E1 21906.113,E2 21906.113} C_VEL
LIN {X 0,Y 623.749,Z 1026.89,A -85,B 0,C 180,E1 21904.741,E2 21904.741} C_VEL
LIN {X 0,Y 621.559,Z 1045.259,A -85,B 0,C 180,E1 21903.268,E2 21903.268} C_VEL
LIN {X 0,Y 619.091,Z 1066.194,A -85,B 0,C 180,E1 21901.39,E2 21901.39} C_VEL
LIN {X 0,Y 616.769,Z 1085.446,A -85,B 0,C 180,E1 21899.42,E2 21899.42} C_VEL
LIN {X 0,Y 615.011,Z 1101.268,A -85,B 0,C 180,E1 21897.616,E2 21897.616} C_VEL
LIN {X 0,Y 613.177,Z 1118.754,A -85,B 0,C 180,E1 21895.392,E2 21895.392} C_VEL
LIN {X 0,Y 611.657,Z 1134.466,A -85,B 0,C 180,E1 21893.1,E2 21893.1} C_VEL
LIN {X 0,Y 610.575,Z 1147.149,A -85,B 0,C 180,E1 21891.017,E2 21891.017} C_VEL
LIN {X 0,Y 609.565,Z 1160.822,A -85,B 0,C 180,E1 21888.457,E2 21888.457} C_VEL
LIN {X 0,Y 608.899,Z 1171.491,A -85,B 0,C 180,E1 21886.112,E2 21886.112} C_VEL
LIN {X 0,Y 608.497,Z 1179.513,A -85,B 0,C 180,E1 21884.075,E2 21884.075} C_VEL
LIN {X 0,Y 608.211,Z 1187.002,A -85,B 0,C 180,E1 21881.859,E2 21881.859} C_VEL
LIN {X 0,Y 608.029,Z 1194.035,A -85,B 0,C 180,E1 21879.274,E2 21879.274} C_VEL
LIN {X 0,Y 607.943,Z 1199.072,A -85,B 0,C 180,E1 21876.801,E2 21876.801} C_VEL
LIN {X 0,Y 607.915,Z 1202.348,A -85,B 0,C 180,E1 21874.528,E2 21874.528} C_VEL
LIN {X 0,Y 607.911,Z 1204.438,A -85,B 0,C 180,E1 21872.074,E2 21872.074} C_VEL
LIN {X 0,Y 607.893,Z 1204.894,A -85,B 0,C 180,E1 21869.529,E2 21869.529} C_VEL
LIN {X 0,Y 607.912,Z 1203.998,A -85,B 0,C 180,E1 21867.266,E2 21867.266} C_VEL
LIN {X 0,Y 607.924,Z 1201.78,A -85,B 0,C 180,E1 21864.999,E2 21864.999} C_VEL
LIN {X 0,Y 607.963,Z 1197.735,A -85,B 0,C 180,E1 21862.44,E2 21862.44} C_VEL
LIN {X 0,Y 608.07,Z 1192.121,A -85,B 0,C 180,E1 21859.962,E2 21859.962} C_VEL
LIN {X 0,Y 608.252,Z 1185.488,A -85,B 0,C 180,E1 21857.661,E2 21857.661} C_VEL
LIN {X 0,Y 608.607,Z 1177.375,A -85,B 0,C 180,E1 21855.345,E2 21855.345} C_VEL
LIN {X 0,Y 609.193,Z 1166.372,A -85,B 0,C 180,E1 21852.718,E2 21852.718} C_VEL
LIN {X 0,Y 609.901,Z 1155.793,A -85,B 0,C 180,E1 21850.562,E2 21850.562} C_VEL
LIN {X 0,Y 610.802,Z 1144.285,A -85,B 0,C 180,E1 21848.489,E2 21848.489} C_VEL
LIN {X 0,Y 612.149,Z 1129.295,A -85,B 0,C 180,E1 21846.104,E2 21846.104} C_VEL
LIN {X 0,Y 613.766,Z 1112.975,A -85,B 0,C 180,E1 21843.85,E2 21843.85} C_VEL
LIN {X 0,Y 615.429,Z 1097.311,A -85,B 0,C 180,E1 21841.911,E2 21841.911} C_VEL
LIN {X 0,Y 617.804,Z 1076.852,A -85,B 0,C 180,E1 21839.672,E2 21839.672} C_VEL
LIN {X 0,Y 619.889,Z 1059.054,A -85,B 0,C 180,E1 21837.949,E2 21837.949} C_VEL
LIN {X 0,Y 621.967,Z 1041.615,A -85,B 0,C 180,E1 21836.426,E2 21836.426} C_VEL
LIN {X 0,Y 624.676,Z 1019.544,A -85,B 0,C 180,E1 21834.703,E2 21834.703} C_VEL
LIN {X 0,Y 627.358,Z 996.428,A -85,B 0,C 180,E1 21833.139,E2 21833.139} C_VEL
LIN {X 0,Y 629.491,Z 977.549,A -85,B 0,C 180,E1 21832.007,E2 21832.007} C_VEL
LIN {X 0,Y 631.516,Z 958.695,A -85,B 0,C 180,E1 21830.998,E2 21830.998} C_VEL
LIN {X 0,Y 633.556,Z 938.332,A -85,B 0,C 180,E1 21830.035,E2 21830.035} C_VEL
LIN {X 0,Y 635.906,Z 913.02,A -85,B 0,C 180,E1 21829.004,E2 21829.004} C_VEL
LIN {X 0,Y 637.95,Z 886.552,A -85,B 0,C 180,E1 21828.131,E2 21828.131} C_VEL
LIN {X 0,Y 639.416,Z 864.711,A -85,B 0,C 180,E1 21827.545,E2 21827.545} C_VEL
LIN {X 0,Y 640.632,Z 842.721,A -85,B 0,C 180,E1 21827.072,E2 21827.072} C_VEL
LIN {X 0,Y 641.728,Z 815.707,A -85,B 0,C 180,E1 21826.638,E2 21826.638} C_VEL
LIN {X 0,Y 646.451,Z 593.381,A -85,B 0,C 180,E1 21823.632,E2 21823.632} C_VEL
LIN {X 0,Y 650.824,Z 401.107,A -85,B 0,C 180,E1 21820.961,E2 21820.961} C_VEL
LIN {X 0,Y 639.782,Z 384.782,A -85,B 0,C 180,E1 21819.53,E2 21819.53} C_VEL
LIN {X 0,Y 630.806,Z 371.728,A -85,B 0,C 180,E1 21818.271,E2 21818.271} C_VEL
LIN {X 0,Y 623.717,Z 361.863,A -85,B 0,C 180,E1 21817.213,E2 21817.213} C_VEL
LIN {X 0,Y 615.821,Z 351.491,A -85,B 0,C 180,E1 21815.97,E2 21815.97} C_VEL
LIN {X 0,Y 614.208,Z 348.993,A -85,B 0,C 180,E1 21815.648,E2 21815.648} C_VEL
LIN {X 0,Y 611.718,Z 344.191,A -85,B 0,C 180,E1 21814.783,E2 21814.783} C_VEL
LIN {X 0,Y 610.925,Z 342.587,A -85,B 0,C 180,E1 21814.492,E2 21814.492} C_VEL
LIN {X 0,Y 609.141,Z 339.12,A -85,B 0,C 180,E1 21813.843,E2 21813.843} C_VEL
LIN {X 0,Y 608.999,Z 338.365,A -85,B 0,C 180,E1 21813.707,E2 21813.707} C_VEL
LIN {X 0,Y 608.994,Z 338.339,A -85,B 0,C 180,E1 21810.925,E2 21810.925} C_VEL
LIN {X 0,Y 608.992,Z 338.356,A -85,B 0,C 180,E1 21807.582,E2 21807.582} C_VEL
LIN {X 0,Y 608.993,Z 338.364,A -85,B 0,C 180,E1 21804.751,E2 21804.751} C_VEL
LIN {X 0,Y 608.983,Z 338.337,A -85,B 0,C 180,E1 21801.419,E2 21801.419} C_VEL
LIN {X 0,Y 608.983,Z 338.373,A -85,B 0,C 180,E1 21798.673,E2 21798.673} C_VEL
LIN {X 0,Y 608.99,Z 338.349,A -85,B 0,C 180,E1 21795.426,E2 21795.426} C_VEL
LIN {X 0,Y 608.971,Z 338.359,A -85,B 0,C 180,E1 21792.71,E2 21792.71} C_VEL
LIN {X 0,Y 609.037,Z 338.352,A -85,B 0,C 180,E1 21789.64,E2 21789.64} C_VEL
LIN {X 0,Y 608.973,Z 338.347,A -85,B 0,C 180,E1 21786.789,E2 21786.789} C_VEL
LIN {X 0,Y 609.038,Z 338.357,A -85,B 0,C 180,E1 21783.86,E2 21783.86} C_VEL
LIN {X 0,Y 608.98,Z 338.336,A -85,B 0,C 180,E1 21780.753,E2 21780.753} C_VEL
LIN {X 0,Y 609.007,Z 338.365,A -85,B 0,C 180,E1 21778.024,E2 21778.024} C_VEL
LIN {X 0,Y 608.996,Z 338.33,A -85,B 0,C 180,E1 21774.819,E2 21774.819} C_VEL
LIN {X 0,Y 609,Z 338.37,A -85,B 0,C 180,E1 21772.073,E2 21772.073} C_VEL
LIN {X 0,Y 609.017,Z 338.336,A -85,B 0,C 180,E1 21768.829,E2 21768.829} C_VEL
LIN {X 0,Y 609.002,Z 338.361,A -85,B 0,C 180,E1 21766.003,E2 21766.003} C_VEL
LIN {X 0,Y 609.039,Z 338.351,A -85,B 0,C 180,E1 21762.811,E2 21762.811} C_VEL
LIN {X 0,Y 609.004,Z 338.336,A -85,B 0,C 180,E1 21759.903,E2 21759.903} C_VEL
LIN {X 0,Y 609.061,Z 338.357,A -85,B 0,C 180,E1 21756.796,E2 21756.796} C_VEL
LIN {X 0,Y 609.011,Z 338.36,A -85,B 0,C 180,E1 21753.791,E2 21753.791} C_VEL
LIN {X 0,Y 609.052,Z 338.488,A -85,B 0,C 180,E1 21751.382,E2 21751.382} C_VEL
LIN {X 0,Y 610.64,Z 342.202,A -85,B 0,C 180,E1 21750.74,E2 21750.74} C_VEL
LIN {X 0,Y 612.707,Z 344.893,A -85,B 0,C 180,E1 21750.392,E2 21750.392} C_VEL
LIN {X 0,Y 616.08,Z 348.791,A -85,B 0,C 180,E1 21749.847,E2 21749.847} C_VEL
LIN {X 0,Y 619.961,Z 353.944,A -85,B 0,C 180,E1 21749.225,E2 21749.225} C_VEL
LIN {X 0,Y 630.978,Z 368.85,A -85,B 0,C 180,E1 21747.56,E2 21747.56} C_VEL
LIN {X 0,Y 645.256,Z 389.382,A -85,B 0,C 180,E1 21745.609,E2 21745.609} C_VEL
LIN {X 0,Y 650.777,Z 398.152,A -85,B 0,C 180,E1 21744.894,E2 21744.894} C_VEL
LIN {X 0,Y 646.685,Z 574.472,A -85,B 0,C 180,E1 21742.446,E2 21742.446} C_VEL
LIN {X 0,Y 645.823,Z 582.175,A -85,B 0,C 180,E1 21742.404,E2 21742.404} C_VEL
LIN {X 0,Y 641.033,Z 602.83,A -85,B 0,C 180,E1 21742.526,E2 21742.526} C_VEL
LIN {X 0,Y 640.352,Z 609.44,A -85,B 0,C 180,E1 21742.485,E2 21742.485} C_VEL
LIN {X 0,Y 635.532,Z 815.902,A -85,B 0,C 180,E1 21739.661,E2 21739.661} C_VEL
LIN {X 0,Y 634.51,Z 837.636,A -85,B 0,C 180,E1 21739.28,E2 21739.28} C_VEL
LIN {X 0,Y 633.117,Z 860.546,A -85,B 0,C 180,E1 21738.759,E2 21738.759} C_VEL
LIN {X 0,Y 631.062,Z 887.962,A -85,B 0,C 180,E1 21737.958,E2 21737.958} C_VEL
LIN {X 0,Y 628.976,Z 911.025,A -85,B 0,C 180,E1 21737.125,E2 21737.125} C_VEL
LIN {X 0,Y 626.959,Z 931.542,A -85,B 0,C 180,E1 21736.256,E2 21736.256} C_VEL
LIN {X 0,Y 624.804,Z 951.715,A -85,B 0,C 180,E1 21735.278,E2 21735.278} C_VEL
LIN {X 0,Y 622.323,Z 973.393,A -85,B 0,C 180,E1 21734.082,E2 21734.082} C_VEL
LIN {X 0,Y 619.277,Z 998.039,A -85,B 0,C 180,E1 21732.508,E2 21732.508} C_VEL
LIN {X 0,Y 616.912,Z 1016.743,A -85,B 0,C 180,E1 21731.149,E2 21731.149} C_VEL
LIN {X 0,Y 614.61,Z 1034.801,A -85,B 0,C 180,E1 21729.69,E2 21729.69} C_VEL
LIN {X 0,Y 612.112,Z 1054.745,A -85,B 0,C 180,E1 21727.893,E2 21727.893} C_VEL
LIN {X 0,Y 609.564,Z 1074.722,A -85,B 0,C 180,E1 21725.844,E2 21725.844} C_VEL
LIN {X 0,Y 607.647,Z 1090.612,A -85,B 0,C 180,E1 21724.018,E2 21724.018} C_VEL
LIN {X 0,Y 605.783,Z 1107.309,A -85,B 0,C 180,E1 21721.882,E2 21721.882} C_VEL
LIN {X 0,Y 604.022,Z 1123.958,A -85,B 0,C 180,E1 21719.448,E2 21719.448} C_VEL
LIN {X 0,Y 602.845,Z 1136.615,A -85,B 0,C 180,E1 21717.35,E2 21717.35} C_VEL
LIN {X 0,Y 601.775,Z 1149.909,A -85,B 0,C 180,E1 21714.857,E2 21714.857} C_VEL
LIN {X 0,Y 600.997,Z 1161.472,A -85,B 0,C 180,E1 21712.291,E2 21712.291} C_VEL
LIN {X 0,Y 600.54,Z 1169.732,A -85,B 0,C 180,E1 21710.16,E2 21710.16} C_VEL
LIN {X 0,Y 600.235,Z 1177.382,A -85,B 0,C 180,E1 21707.848,E2 21707.848} C_VEL
LIN {X 0,Y 600.03,Z 1184.464,A -85,B 0,C 180,E1 21705.166,E2 21705.166} C_VEL
LIN {X 0,Y 599.945,Z 1189.138,A -85,B 0,C 180,E1 21702.806,E2 21702.806} C_VEL
LIN {X 0,Y 599.917,Z 1192.438,A -85,B 0,C 180,E1 21700.465,E2 21700.465} C_VEL
LIN {X 0,Y 599.911,Z 1194.499,A -85,B 0,C 180,E1 21697.951,E2 21697.951} C_VEL
LIN {X 0,Y 599.895,Z 1194.888,A -85,B 0,C 180,E1 21695.451,E2 21695.451} C_VEL
LIN {X 0,Y 599.911,Z 1194.041,A -85,B 0,C 180,E1 21693.248,E2 21693.248} C_VEL
LIN {X 0,Y 599.923,Z 1191.858,A -85,B 0,C 180,E1 21690.955,E2 21690.955} C_VEL
LIN {X 0,Y 599.961,Z 1188.055,A -85,B 0,C 180,E1 21688.472,E2 21688.472} C_VEL
LIN {X 0,Y 600.079,Z 1182.4,A -85,B 0,C 180,E1 21685.891,E2 21685.891} C_VEL
LIN {X 0,Y 600.296,Z 1175.63,A -85,B 0,C 180,E1 21683.496,E2 21683.496} C_VEL
LIN {X 0,Y 600.653,Z 1167.703,A -85,B 0,C 180,E1 21681.19,E2 21681.19} C_VEL
LIN {X 0,Y 601.272,Z 1157.045,A -85,B 0,C 180,E1 21678.586,E2 21678.586} C_VEL
LIN {X 0,Y 602.079,Z 1145.832,A -85,B 0,C 180,E1 21676.262,E2 21676.262} C_VEL
LIN {X 0,Y 603.087,Z 1133.831,A -85,B 0,C 180,E1 21674.074,E2 21674.074} C_VEL
LIN {X 0,Y 604.68,Z 1117.559,A -85,B 0,C 180,E1 21671.489,E2 21671.489} C_VEL
LIN {X 0,Y 606.238,Z 1102.813,A -85,B 0,C 180,E1 21669.433,E2 21669.433} C_VEL
LIN {X 0,Y 608.068,Z 1087.135,A -85,B 0,C 180,E1 21667.472,E2 21667.472} C_VEL
LIN {X 0,Y 610.568,Z 1066.698,A -85,B 0,C 180,E1 21665.214,E2 21665.214} C_VEL
LIN {X 0,Y 612.707,Z 1049.651,A -85,B 0,C 180,E1 21663.544,E2 21663.544} C_VEL
LIN {X 0,Y 614.821,Z 1033.051,A -85,B 0,C 180,E1 21662.071,E2 21662.071} C_VEL
LIN {X 0,Y 617.26,Z 1014.047,A -85,B 0,C 180,E1 21660.552,E2 21660.552} C_VEL
LIN {X 0,Y 620.445,Z 988.919,A -85,B 0,C 180,E1 21658.794,E2 21658.794} C_VEL
LIN {X 0,Y 622.837,Z 968.96,A -85,B 0,C 180,E1 21657.575,E2 21657.575} C_VEL
LIN {X 0,Y 624.98,Z 950.166,A -85,B 0,C 180,E1 21656.554,E2 21656.554} C_VEL
LIN {X 0,Y 627.013,Z 931.037,A -85,B 0,C 180,E1 21655.631,E2 21655.631} C_VEL
LIN {X 0,Y 629.04,Z 910.388,A -85,B 0,C 180,E1 21654.76,E2 21654.76} C_VEL
LIN {X 0,Y 631.343,Z 885.02,A -85,B 0,C 180,E1 21653.853,E2 21653.853} C_VEL
LIN {X 0,Y 633.23,Z 858.738,A -85,B 0,C 180,E1 21653.107,E2 21653.107} C_VEL
LIN {X 0,Y 634.542,Z 836.933,A -85,B 0,C 180,E1 21652.616,E2 21652.616} C_VEL
LIN {X 0,Y 635.557,Z 815.181,A -85,B 0,C 180,E1 21652.238,E2 21652.238} C_VEL
LIN {X 0,Y 640.467,Z 604.546,A -85,B 0,C 180,E1 21649.358,E2 21649.358} C_VEL
LIN {X 0,Y 645.413,Z 401.64,A -85,B 0,C 180,E1 21646.524,E2 21646.524} C_VEL
LIN {X 0,Y 632.776,Z 383.081,A -85,B 0,C 180,E1 21644.842,E2 21644.842} C_VEL
LIN {X 0,Y 619.44,Z 364.91,A -85,B 0,C 180,E1 21643,E2 21643} C_VEL
LIN {X 0,Y 611.073,Z 353.859,A -85,B 0,C 180,E1 21641.788,E2 21641.788} C_VEL
LIN {X 0,Y 605.953,Z 347.225,A -85,B 0,C 180,E1 21641.021,E2 21641.021} C_VEL
LIN {X 0,Y 603.825,Z 344.416,A -85,B 0,C 180,E1 21640.694,E2 21640.694} C_VEL
LIN {X 0,Y 601.878,Z 341.921,A -85,B 0,C 180,E1 21640.384,E2 21640.384} C_VEL
LIN {X 0,Y 601.113,Z 339.356,A -85,B 0,C 180,E1 21639.982,E2 21639.982} C_VEL
LIN {X 0,Y 601.124,Z 339.359,A -85,B 0,C 180,E1 21636.666,E2 21636.666} C_VEL
LIN {X 0,Y 601.125,Z 339.347,A -85,B 0,C 180,E1 21633.521,E2 21633.521} C_VEL
LIN {X 0,Y 601.099,Z 339.349,A -85,B 0,C 180,E1 21630.267,E2 21630.267} C_VEL
LIN {X 0,Y 601.135,Z 339.31,A -85,B 0,C 180,E1 21627.142,E2 21627.142} C_VEL
LIN {X 0,Y 601.089,Z 339.356,A -85,B 0,C 180,E1 21623.947,E2 21623.947} C_VEL
LIN {X 0,Y 601.137,Z 339.303,A -85,B 0,C 180,E1 21620.807,E2 21620.807} C_VEL
LIN {X 0,Y 601.083,Z 339.355,A -85,B 0,C 180,E1 21617.723,E2 21617.723} C_VEL
LIN {X 0,Y 601.135,Z 339.303,A -85,B 0,C 180,E1 21614.546,E2 21614.546} C_VEL
LIN {X 0,Y 601.075,Z 339.35,A -85,B 0,C 180,E1 21611.515,E2 21611.515} C_VEL
LIN {X 0,Y 601.125,Z 339.342,A -85,B 0,C 180,E1 21608.321,E2 21608.321} C_VEL
LIN {X 0,Y 601.066,Z 339.346,A -85,B 0,C 180,E1 21605.345,E2 21605.345} C_VEL
LIN {X 0,Y 601.118,Z 339.344,A -85,B 0,C 180,E1 21602.193,E2 21602.193} C_VEL
LIN {X 0,Y 601.061,Z 339.356,A -85,B 0,C 180,E1 21599.237,E2 21599.237} C_VEL
LIN {X 0,Y 601.115,Z 339.354,A -85,B 0,C 180,E1 21596.089,E2 21596.089} C_VEL
LIN {X 0,Y 601.053,Z 339.359,A -85,B 0,C 180,E1 21593.121,E2 21593.121} C_VEL
LIN {X 0,Y 601.12,Z 339.352,A -85,B 0,C 180,E1 21590.038,E2 21590.038} C_VEL
LIN {X 0,Y 601.04,Z 339.318,A -85,B 0,C 180,E1 21587.021,E2 21587.021} C_VEL
LIN {X 0,Y 601.121,Z 339.347,A -85,B 0,C 180,E1 21583.971,E2 21583.971} C_VEL
LIN {X 0,Y 601.033,Z 339.32,A -85,B 0,C 180,E1 21580.896,E2 21580.896} C_VEL
LIN {X 0,Y 601.116,Z 339.353,A -85,B 0,C 180,E1 21577.815,E2 21577.815} C_VEL
LIN {X 0,Y 601.028,Z 339.315,A -85,B 0,C 180,E1 21574.793,E2 21574.793} C_VEL
LIN {X 0,Y 601.117,Z 339.349,A -85,B 0,C 180,E1 21571.701,E2 21571.701} C_VEL
LIN {X 0,Y 601.04,Z 339.353,A -85,B 0,C 180,E1 21568.732,E2 21568.732} C_VEL
LIN {X 0,Y 601.075,Z 339.567,A -85,B 0,C 180,E1 21566.704,E2 21566.704} C_VEL
LIN {X 0,Y 602.297,Z 342.74,A -85,B 0,C 180,E1 21566.21,E2 21566.21} C_VEL
LIN {X 0,Y 603.588,Z 344.74,A -85,B 0,C 180,E1 21565.835,E2 21565.835} C_VEL
LIN {X 0,Y 606.196,Z 350.08,A -85,B 0,C 180,E1 21564.998,E2 21564.998} C_VEL
LIN {X 0,Y 617.868,Z 365.767,A -85,B 0,C 180,E1 21563.276,E2 21563.276} C_VEL
LIN {X 0,Y 630.662,Z 383.062,A -85,B 0,C 180,E1 21561.501,E2 21561.501} C_VEL
LIN {X 0,Y 645.49,Z 404.969,A -85,B 0,C 180,E1 21559.522,E2 21559.522} C_VEL
LIN {X 0,Y 640.659,Z 604.663,A -85,B 0,C 180,E1 21556.731,E2 21556.731} C_VEL
LIN {X 0,Y 635.656,Z 822.502,A -85,B 0,C 180,E1 21553.757,E2 21553.757} C_VEL
LIN {X 0,Y 634.662,Z 844.609,A -85,B 0,C 180,E1 21553.385,E2 21553.385} C_VEL
LIN {X 0,Y 633.401,Z 865.986,A -85,B 0,C 180,E1 21552.917,E2 21552.917} C_VEL
LIN {X 0,Y 631.749,Z 889.195,A -85,B 0,C 180,E1 21552.281,E2 21552.281} C_VEL
LIN {X 0,Y 629.337,Z 917.421,A -85,B 0,C 180,E1 21551.311,E2 21551.311} C_VEL
LIN {X 0,Y 627.187,Z 939.438,A -85,B 0,C 180,E1 21550.395,E2 21550.395} C_VEL
LIN {X 0,Y 625.15,Z 958.67,A -85,B 0,C 180,E1 21549.477,E2 21549.477} C_VEL
LIN {X 0,Y 622.994,Z 977.623,A -85,B 0,C 180,E1 21548.457,E2 21548.457} C_VEL
LIN {X 0,Y 620.636,Z 997.346,A -85,B 0,C 180,E1 21547.262,E2 21547.262} C_VEL
LIN {X 0,Y 617.614,Z 1021.547,A -85,B 0,C 180,E1 21545.592,E2 21545.592} C_VEL
LIN {X 0,Y 614.968,Z 1041.906,A -85,B 0,C 180,E1 21543.981,E2 21543.981} C_VEL
LIN {X 0,Y 612.786,Z 1059.044,A -85,B 0,C 180,E1 21542.468,E2 21542.468} C_VEL
LIN {X 0,Y 610.53,Z 1077.073,A -85,B 0,C 180,E1 21540.704,E2 21540.704} C_VEL
LIN {X 0,Y 608.06,Z 1097.142,A -85,B 0,C 180,E1 21538.481,E2 21538.481} C_VEL
LIN {X 0,Y 606.26,Z 1112.612,A -85,B 0,C 180,E1 21536.548,E2 21536.548} C_VEL
LIN {X 0,Y 604.641,Z 1127.885,A -85,B 0,C 180,E1 21534.42,E2 21534.42} C_VEL
LIN {X 0,Y 603.102,Z 1143.697,A -85,B 0,C 180,E1 21531.903,E2 21531.903} C_VEL
LIN {X 0,Y 602.122,Z 1155.269,A -85,B 0,C 180,E1 21529.802,E2 21529.802} C_VEL
LIN {X 0,Y 601.342,Z 1165.906,A -85,B 0,C 180,E1 21527.615,E2 21527.615} C_VEL
LIN {X 0,Y 600.69,Z 1177.017,A -85,B 0,C 180,E1 21524.952,E2 21524.952} C_VEL
LIN {X 0,Y 600.298,Z 1185.324,A -85,B 0,C 180,E1 21522.557,E2 21522.557} C_VEL
LIN {X 0,Y 600.092,Z 1191.862,A -85,B 0,C 180,E1 21520.27,E2 21520.27} C_VEL
LIN {X 0,Y 599.973,Z 1197.542,A -85,B 0,C 180,E1 21517.758,E2 21517.758} C_VEL
LIN {X 0,Y 599.927,Z 1201.663,A -85,B 0,C 180,E1 21515.164,E2 21515.164} C_VEL
LIN {X 0,Y 599.915,Z 1203.927,A -85,B 0,C 180,E1 21512.866,E2 21512.866} C_VEL
LIN {X 0,Y 599.895,Z 1204.849,A -85,B 0,C 180,E1 21510.669,E2 21510.669} C_VEL
LIN {X 0,Y 599.908,Z 1204.623,A -85,B 0,C 180,E1 21508.377,E2 21508.377} C_VEL
LIN {X 0,Y 599.918,Z 1202.789,A -85,B 0,C 180,E1 21505.795,E2 21505.795} C_VEL
LIN {X 0,Y 599.944,Z 1199.513,A -85,B 0,C 180,E1 21503.375,E2 21503.375} C_VEL
LIN {X 0,Y 600.014,Z 1195.106,A -85,B 0,C 180,E1 21501.085,E2 21501.085} C_VEL
LIN {X 0,Y 600.197,Z 1188.477,A -85,B 0,C 180,E1 21498.469,E2 21498.469} C_VEL
LIN {X 0,Y 600.504,Z 1180.573,A -85,B 0,C 180,E1 21496.029,E2 21496.029} C_VEL
LIN {X 0,Y 600.938,Z 1172.307,A -85,B 0,C 180,E1 21493.868,E2 21493.868} C_VEL
LIN {X 0,Y 601.567,Z 1162.693,A -85,B 0,C 180,E1 21491.692,E2 21491.692} C_VEL
LIN {X 0,Y 602.621,Z 1149.398,A -85,B 0,C 180,E1 21489.092,E2 21489.092} C_VEL
LIN {X 0,Y 603.844,Z 1135.74,A -85,B 0,C 180,E1 21486.791,E2 21486.791} C_VEL
LIN {X 0,Y 605.279,Z 1121.577,A -85,B 0,C 180,E1 21484.669,E2 21484.669} C_VEL
LIN {X 0,Y 607.374,Z 1103.065,A -85,B 0,C 180,E1 21482.233,E2 21482.233} C_VEL
LIN {X 0,Y 609.274,Z 1086.963,A -85,B 0,C 180,E1 21480.359,E2 21480.359} C_VEL
LIN {X 0,Y 611.357,Z 1070.396,A -85,B 0,C 180,E1 21478.622,E2 21478.622} C_VEL
LIN {X 0,Y 614.091,Z 1049.295,A -85,B 0,C 180,E1 21476.646,E2 21476.646} C_VEL
LIN {X 0,Y 616.658,Z 1028.868,A -85,B 0,C 180,E1 21474.969,E2 21474.969} C_VEL
LIN {X 0,Y 619.039,Z 1009.974,A -85,B 0,C 180,E1 21473.583,E2 21473.583} C_VEL
LIN {X 0,Y 621.633,Z 988.939,A -85,B 0,C 180,E1 21472.206,E2 21472.206} C_VEL
LIN {X 0,Y 624.589,Z 963.715,A -85,B 0,C 180,E1 21470.778,E2 21470.778} C_VEL
LIN {X 0,Y 626.82,Z 942.851,A -85,B 0,C 180,E1 21469.757,E2 21469.757} C_VEL
LIN {X 0,Y 628.831,Z 922.578,A -85,B 0,C 180,E1 21468.892,E2 21468.892} C_VEL
LIN {X 0,Y 630.688,Z 901.893,A -85,B 0,C 180,E1 21468.131,E2 21468.131} C_VEL
LIN {X 0,Y 632.496,Z 879.248,A -85,B 0,C 180,E1 21467.429,E2 21467.429} C_VEL
LIN {X 0,Y 634.364,Z 850.596,A -85,B 0,C 180,E1 21466.732,E2 21466.732} C_VEL
LIN {X 0,Y 635.498,Z 826.736,A -85,B 0,C 180,E1 21466.306,E2 21466.306} C_VEL
LIN {X 0,Y 640.109,Z 628.386,A -85,B 0,C 180,E1 21463.596,E2 21463.596} C_VEL
LIN {X 0,Y 645.094,Z 421.33,A -85,B 0,C 180,E1 21460.712,E2 21460.712} C_VEL
LIN {X 0,Y 645.375,Z 404.812,A -85,B 0,C 180,E1 21460.464,E2 21460.464} C_VEL
LIN {X 0,Y 630.127,Z 382.027,A -85,B 0,C 180,E1 21458.38,E2 21458.38} C_VEL
LIN {X 0,Y 620.188,Z 368.125,A -85,B 0,C 180,E1 21456.881,E2 21456.881} C_VEL
LIN {X 0,Y 609.816,Z 354.302,A -85,B 0,C 180,E1 21455.194,E2 21455.194} C_VEL
LIN {X 0,Y 606.43,Z 349.929,A -85,B 0,C 180,E1 21454.612,E2 21454.612} C_VEL
LIN {X 0,Y 605.302,Z 348.049,A -85,B 0,C 180,E1 21454.284,E2 21454.284} C_VEL
LIN {X 0,Y 603.229,Z 343.915,A -85,B 0,C 180,E1 21453.502,E2 21453.502} C_VEL
LIN {X 0,Y 601.338,Z 340.632,A -85,B 0,C 180,E1 21452.825,E2 21452.825} C_VEL
LIN {X 0,Y 601.098,Z 339.358,A -85,B 0,C 180,E1 21452.613,E2 21452.613} C_VEL
LIN {X 0,Y 601.047,Z 339.339,A -85,B 0,C 180,E1 21449.5,E2 21449.5} C_VEL
LIN {X 0,Y 601.054,Z 339.326,A -85,B 0,C 180,E1 21446.797,E2 21446.797} C_VEL
LIN {X 0,Y 601.054,Z 339.357,A -85,B 0,C 180,E1 21443.532,E2 21443.532} C_VEL
LIN {X 0,Y 601.036,Z 339.331,A -85,B 0,C 180,E1 21440.856,E2 21440.856} C_VEL
LIN {X 0,Y 601.081,Z 339.332,A -85,B 0,C 180,E1 21437.723,E2 21437.723} C_VEL
LIN {X 0,Y 601.03,Z 339.357,A -85,B 0,C 180,E1 21434.845,E2 21434.845} C_VEL
LIN {X 0,Y 601.106,Z 339.316,A -85,B 0,C 180,E1 21431.806,E2 21431.806} C_VEL
LIN {X 0,Y 601.034,Z 339.362,A -85,B 0,C 180,E1 21428.804,E2 21428.804} C_VEL
LIN {X 0,Y 601.096,Z 339.315,A -85,B 0,C 180,E1 21425.892,E2 21425.892} C_VEL
LIN {X 0,Y 601.044,Z 339.36,A -85,B 0,C 180,E1 21422.765,E2 21422.765} C_VEL
LIN {X 0,Y 601.093,Z 339.316,A -85,B 0,C 180,E1 21419.809,E2 21419.809} C_VEL
LIN {X 0,Y 601.05,Z 339.355,A -85,B 0,C 180,E1 21416.662,E2 21416.662} C_VEL
LIN {X 0,Y 601.095,Z 339.326,A -85,B 0,C 180,E1 21413.697,E2 21413.697} C_VEL
LIN {X 0,Y 601.056,Z 339.336,A -85,B 0,C 180,E1 21410.562,E2 21410.562} C_VEL
LIN {X 0,Y 601.098,Z 339.345,A -85,B 0,C 180,E1 21407.609,E2 21407.609} C_VEL
LIN {X 0,Y 601.062,Z 339.317,A -85,B 0,C 180,E1 21404.465,E2 21404.465} C_VEL
LIN {X 0,Y 601.092,Z 339.354,A -85,B 0,C 180,E1 21401.575,E2 21401.575} C_VEL
LIN {X 0,Y 601.068,Z 339.34,A -85,B 0,C 180,E1 21398.327,E2 21398.327} C_VEL
LIN {X 0,Y 601.088,Z 339.322,A -85,B 0,C 180,E1 21395.491,E2 21395.491} C_VEL
LIN {X 0,Y 601.113,Z 339.441,A -85,B 0,C 180,E1 21392.488,E2 21392.488} C_VEL
LIN {X 0,Y 602.332,Z 342.769,A -85,B 0,C 180,E1 21391.952,E2 21391.952} C_VEL
LIN {X 0,Y 605.19,Z 345.998,A -85,B 0,C 180,E1 21391.452,E2 21391.452} C_VEL
LIN {X 0,Y 609.748,Z 351.791,A -85,B 0,C 180,E1 21390.666,E2 21390.666} C_VEL
LIN {X 0,Y 614.051,Z 357.207,A -85,B 0,C 180,E1 21389.952,E2 21389.952} C_VEL
LIN {X 0,Y 618.423,Z 363.005,A -85,B 0,C 180,E1 21389.248,E2 21389.248} C_VEL
LIN {X 0,Y 626.396,Z 373.737,A -85,B 0,C 180,E1 21388.024,E2 21388.024} C_VEL
LIN {X 0,Y 638.8,Z 391.81,A -85,B 0,C 180,E1 21386.257,E2 21386.257} C_VEL
LIN {X 0,Y 645.434,Z 401.999,A -85,B 0,C 180,E1 21385.378,E2 21385.378} C_VEL
LIN {X 0,Y 640.352,Z 609.44,A -85,B 0,C 180,E1 21382.485,E2 21382.485} C_VEL
LIN {X 0,Y 639.471,Z 617.146,A -85,B 0,C 180,E1 21382.445,E2 21382.445} C_VEL
LIN {X 0,Y 634.649,Z 637.796,A -85,B 0,C 180,E1 21382.572,E2 21382.572} C_VEL
LIN {X 0,Y 633.986,Z 644.403,A -85,B 0,C 180,E1 21382.528,E2 21382.528} C_VEL
LIN {X 0,Y 629.708,Z 817.004,A -85,B 0,C 180,E1 21380.149,E2 21380.149} C_VEL
LIN {X 0,Y 628.586,Z 839.377,A -85,B 0,C 180,E1 21379.749,E2 21379.749} C_VEL
LIN {X 0,Y 626.85,Z 866.105,A -85,B 0,C 180,E1 21379.118,E2 21379.118} C_VEL
LIN {X 0,Y 624.71,Z 891.495,A -85,B 0,C 180,E1 21378.335,E2 21378.335} C_VEL
LIN {X 0,Y 622.694,Z 912.665,A -85,B 0,C 180,E1 21377.553,E2 21377.553} C_VEL
LIN {X 0,Y 620.502,Z 933.659,A -85,B 0,C 180,E1 21376.649,E2 21376.649} C_VEL
LIN {X 0,Y 617.827,Z 957.229,A -85,B 0,C 180,E1 21375.477,E2 21375.477} C_VEL
LIN {X 0,Y 614.723,Z 981.918,A -85,B 0,C 180,E1 21374.032,E2 21374.032} C_VEL
LIN {X 0,Y 612.174,Z 1001.356,A -85,B 0,C 180,E1 21372.737,E2 21372.737} C_VEL
LIN {X 0,Y 609.717,Z 1019.752,A -85,B 0,C 180,E1 21371.366,E2 21371.366} C_VEL
LIN {X 0,Y 606.807,Z 1041.607,A -85,B 0,C 180,E1 21369.541,E2 21369.541} C_VEL
LIN {X 0,Y 604.071,Z 1061.409,A -85,B 0,C 180,E1 21367.645,E2 21367.645} C_VEL
LIN {X 0,Y 601.878,Z 1077.759,A -85,B 0,C 180,E1 21365.903,E2 21365.903} C_VEL
LIN {X 0,Y 599.721,Z 1095.155,A -85,B 0,C 180,E1 21363.838,E2 21363.838} C_VEL
LIN {X 0,Y 597.593,Z 1112.694,A -85,B 0,C 180,E1 21361.468,E2 21361.468} C_VEL
LIN {X 0,Y 596.138,Z 1126.029,A -85,B 0,C 180,E1 21359.434,E2 21359.434} C_VEL
LIN {X 0,Y 594.81,Z 1139.672,A -85,B 0,C 180,E1 21357.1,E2 21357.1} C_VEL
LIN {X 0,Y 593.683,Z 1152.882,A -85,B 0,C 180,E1 21354.475,E2 21354.475} C_VEL
LIN {X 0,Y 593.032,Z 1162.369,A -85,B 0,C 180,E1 21352.294,E2 21352.294} C_VEL
LIN {X 0,Y 592.559,Z 1170.511,A -85,B 0,C 180,E1 21350.134,E2 21350.134} C_VEL
LIN {X 0,Y 592.236,Z 1178.332,A -85,B 0,C 180,E1 21347.691,E2 21347.691} C_VEL
LIN {X 0,Y 592.027,Z 1184.929,A -85,B 0,C 180,E1 21345.075,E2 21345.075} C_VEL
LIN {X 0,Y 591.944,Z 1189.486,A -85,B 0,C 180,E1 21342.684,E2 21342.684} C_VEL
LIN {X 0,Y 591.919,Z 1192.682,A -85,B 0,C 180,E1 21340.314,E2 21340.314} C_VEL
LIN {X 0,Y 591.907,Z 1194.607,A -85,B 0,C 180,E1 21337.669,E2 21337.669} C_VEL
LIN {X 0,Y 591.9,Z 1194.862,A -85,B 0,C 180,E1 21335.331,E2 21335.331} C_VEL
LIN {X 0,Y 591.912,Z 1193.959,A -85,B 0,C 180,E1 21333.098,E2 21333.098} C_VEL
LIN {X 0,Y 591.924,Z 1191.723,A -85,B 0,C 180,E1 21330.774,E2 21330.774} C_VEL
LIN {X 0,Y 591.975,Z 1187.679,A -85,B 0,C 180,E1 21328.161,E2 21328.161} C_VEL
LIN {X 0,Y 592.101,Z 1182.107,A -85,B 0,C 180,E1 21325.641,E2 21325.641} C_VEL
LIN {X 0,Y 592.334,Z 1175.581,A -85,B 0,C 180,E1 21323.311,E2 21323.311} C_VEL
LIN {X 0,Y 592.731,Z 1167.302,A -85,B 0,C 180,E1 21320.876,E2 21320.876} C_VEL
LIN {X 0,Y 593.431,Z 1156.475,A -85,B 0,C 180,E1 21318.223,E2 21318.223} C_VEL
LIN {X 0,Y 594.259,Z 1145.761,A -85,B 0,C 180,E1 21315.978,E2 21315.978} C_VEL
LIN {X 0,Y 595.328,Z 1134.039,A -85,B 0,C 180,E1 21313.811,E2 21313.811} C_VEL
LIN {X 0,Y 597.005,Z 1118.143,A -85,B 0,C 180,E1 21311.242,E2 21311.242} C_VEL
LIN {X 0,Y 598.651,Z 1103.457,A -85,B 0,C 180,E1 21309.16,E2 21309.16} C_VEL
LIN {X 0,Y 600.61,Z 1087.843,A -85,B 0,C 180,E1 21307.176,E2 21307.176} C_VEL
LIN {X 0,Y 603.254,Z 1067.542,A -85,B 0,C 180,E1 21304.893,E2 21304.893} C_VEL
LIN {X 0,Y 605.659,Z 1049.513,A -85,B 0,C 180,E1 21303.106,E2 21303.106} C_VEL
LIN {X 0,Y 607.986,Z 1032.366,A -85,B 0,C 180,E1 21301.573,E2 21301.573} C_VEL
LIN {X 0,Y 610.81,Z 1011.962,A -85,B 0,C 180,E1 21299.939,E2 21299.939} C_VEL
LIN {X 0,Y 613.881,Z 988.703,A -85,B 0,C 180,E1 21298.313,E2 21298.313} C_VEL
LIN {X 0,Y 616.412,Z 968.715,A -85,B 0,C 180,E1 21297.084,E2 21297.084} C_VEL
LIN {X 0,Y 618.684,Z 949.884,A -85,B 0,C 180,E1 21296.056,E2 21296.056} C_VEL
LIN {X 0,Y 620.836,Z 930.712,A -85,B 0,C 180,E1 21295.128,E2 21295.128} C_VEL
LIN {X 0,Y 623.092,Z 908.801,A -85,B 0,C 180,E1 21294.203,E2 21294.203} C_VEL
LIN {X 0,Y 625.656,Z 880.735,A -85,B 0,C 180,E1 21293.223,E2 21293.223} C_VEL
LIN {X 0,Y 627.413,Z 857.485,A -85,B 0,C 180,E1 21292.574,E2 21292.574} C_VEL
LIN {X 0,Y 628.748,Z 836.291,A -85,B 0,C 180,E1 21292.099,E2 21292.099} C_VEL
LIN {X 0,Y 629.814,Z 814.335,A -85,B 0,C 180,E1 21291.72,E2 21291.72} C_VEL
LIN {X 0,Y 635.093,Z 599.694,A -85,B 0,C 180,E1 21288.763,E2 21288.763} C_VEL
LIN {X 0,Y 640.103,Z 405.59,A -85,B 0,C 180,E1 21286.032,E2 21286.032} C_VEL
LIN {X 0,Y 626.661,Z 385.855,A -85,B 0,C 180,E1 21284.209,E2 21284.209} C_VEL
LIN {X 0,Y 611.389,Z 365.35,A -85,B 0,C 180,E1 21282.045,E2 21282.045} C_VEL
LIN {X 0,Y 602.649,Z 353.822,A -85,B 0,C 180,E1 21280.728,E2 21280.728} C_VEL
LIN {X 0,Y 596.334,Z 345.761,A -85,B 0,C 180,E1 21279.736,E2 21279.736} C_VEL
LIN {X 0,Y 593.989,Z 342.949,A -85,B 0,C 180,E1 21279.361,E2 21279.361} C_VEL
LIN {X 0,Y 593.417,Z 341.464,A -85,B 0,C 180,E1 21279.188,E2 21279.188} C_VEL
LIN {X 0,Y 593.199,Z 340.343,A -85,B 0,C 180,E1 21279.009,E2 21279.009} C_VEL
LIN {X 0,Y 593.172,Z 340.338,A -85,B 0,C 180,E1 21275.798,E2 21275.798} C_VEL
LIN {X 0,Y 593.169,Z 340.342,A -85,B 0,C 180,E1 21272.415,E2 21272.415} C_VEL
LIN {X 0,Y 593.2,Z 340.339,A -85,B 0,C 180,E1 21269.263,E2 21269.263} C_VEL
LIN {X 0,Y 593.149,Z 340.297,A -85,B 0,C 180,E1 21266.04,E2 21266.04} C_VEL
LIN {X 0,Y 593.201,Z 340.338,A -85,B 0,C 180,E1 21262.915,E2 21262.915} C_VEL
LIN {X 0,Y 593.139,Z 340.297,A -85,B 0,C 180,E1 21259.806,E2 21259.806} C_VEL
LIN {X 0,Y 593.201,Z 340.339,A -85,B 0,C 180,E1 21256.652,E2 21256.652} C_VEL
LIN {X 0,Y 593.133,Z 340.289,A -85,B 0,C 180,E1 21253.552,E2 21253.552} C_VEL
LIN {X 0,Y 593.189,Z 340.344,A -85,B 0,C 180,E1 21250.391,E2 21250.391} C_VEL
LIN {X 0,Y 593.133,Z 340.344,A -85,B 0,C 180,E1 21247.361,E2 21247.361} C_VEL
LIN {X 0,Y 593.171,Z 340.337,A -85,B 0,C 180,E1 21244.157,E2 21244.157} C_VEL
LIN {X 0,Y 593.128,Z 340.336,A -85,B 0,C 180,E1 21241.159,E2 21241.159} C_VEL
LIN {X 0,Y 593.158,Z 340.333,A -85,B 0,C 180,E1 21237.971,E2 21237.971} C_VEL
LIN {X 0,Y 593.119,Z 340.339,A -85,B 0,C 180,E1 21235.068,E2 21235.068} C_VEL
LIN {X 0,Y 593.153,Z 340.335,A -85,B 0,C 180,E1 21231.859,E2 21231.859} C_VEL
LIN {X 0,Y 593.113,Z 340.347,A -85,B 0,C 180,E1 21228.92,E2 21228.92} C_VEL
LIN {X 0,Y 593.145,Z 340.298,A -85,B 0,C 180,E1 21225.752,E2 21225.752} C_VEL
LIN {X 0,Y 593.102,Z 340.35,A -85,B 0,C 180,E1 21222.841,E2 21222.841} C_VEL
LIN {X 0,Y 593.144,Z 340.3,A -85,B 0,C 180,E1 21219.68,E2 21219.68} C_VEL
LIN {X 0,Y 593.093,Z 340.349,A -85,B 0,C 180,E1 21216.87,E2 21216.87} C_VEL
LIN {X 0,Y 593.166,Z 340.304,A -85,B 0,C 180,E1 21213.737,E2 21213.737} C_VEL
LIN {X 0,Y 593.097,Z 340.343,A -85,B 0,C 180,E1 21210.731,E2 21210.731} C_VEL
LIN {X 0,Y 593.195,Z 340.447,A -85,B 0,C 180,E1 21207.685,E2 21207.685} C_VEL
LIN {X 0,Y 594.277,Z 343.581,A -85,B 0,C 180,E1 21207.195,E2 21207.195} C_VEL
LIN {X 0,Y 595.546,Z 345.513,A -85,B 0,C 180,E1 21206.815,E2 21206.815} C_VEL
LIN {X 0,Y 597.548,Z 349.407,A -85,B 0,C 180,E1 21206.136,E2 21206.136} C_VEL
LIN {X 0,Y 601.545,Z 354.815,A -85,B 0,C 180,E1 21205.5,E2 21205.5} C_VEL
LIN {X 0,Y 617.993,Z 377.069,A -85,B 0,C 180,E1 21203.053,E2 21203.053} C_VEL
LIN {X 0,Y 630.574,Z 394.682,A -85,B 0,C 180,E1 21201.306,E2 21201.306} C_VEL
LIN {X 0,Y 640.194,Z 409.108,A -85,B 0,C 180,E1 21200.008,E2 21200.008} C_VEL
LIN {X 0,Y 634.98,Z 612.229,A -85,B 0,C 180,E1 21197.153,E2 21197.153} C_VEL
LIN {X 0,Y 629.79,Z 824.523,A -85,B 0,C 180,E1 21194.23,E2 21194.23} C_VEL
LIN {X 0,Y 628.738,Z 846.318,A -85,B 0,C 180,E1 21193.854,E2 21193.854} C_VEL
LIN {X 0,Y 627.333,Z 868.736,A -85,B 0,C 180,E1 21193.35,E2 21193.35} C_VEL
LIN {X 0,Y 625.235,Z 895.947,A -85,B 0,C 180,E1 21192.568,E2 21192.568} C_VEL
LIN {X 0,Y 623.05,Z 919.236,A -85,B 0,C 180,E1 21191.733,E2 21191.733} C_VEL
LIN {X 0,Y 620.98,Z 939.435,A -85,B 0,C 180,E1 21190.884,E2 21190.884} C_VEL
LIN {X 0,Y 618.826,Z 958.667,A -85,B 0,C 180,E1 21189.961,E2 21189.961} C_VEL
LIN {X 0,Y 616.546,Z 977.619,A -85,B 0,C 180,E1 21188.934,E2 21188.934} C_VEL
LIN {X 0,Y 614.091,Z 997.043,A -85,B 0,C 180,E1 21187.75,E2 21187.75} C_VEL
LIN {X 0,Y 610.967,Z 1020.877,A -85,B 0,C 180,E1 21186.097,E2 21186.097} C_VEL
LIN {X 0,Y 608.095,Z 1041.606,A -85,B 0,C 180,E1 21184.446,E2 21184.446} C_VEL
LIN {X 0,Y 605.721,Z 1059.043,A -85,B 0,C 180,E1 21182.894,E2 21182.894} C_VEL
LIN {X 0,Y 603.289,Z 1077.265,A -85,B 0,C 180,E1 21181.092,E2 21181.092} C_VEL
LIN {X 0,Y 600.701,Z 1097.14,A -85,B 0,C 180,E1 21178.863,E2 21178.863} C_VEL
LIN {X 0,Y 598.746,Z 1112.644,A -85,B 0,C 180,E1 21176.903,E2 21176.903} C_VEL
LIN {X 0,Y 597.074,Z 1127.451,A -85,B 0,C 180,E1 21174.815,E2 21174.815} C_VEL
LIN {X 0,Y 595.364,Z 1143.699,A -85,B 0,C 180,E1 21172.202,E2 21172.202} C_VEL
LIN {X 0,Y 594.3,Z 1155.267,A -85,B 0,C 180,E1 21170.073,E2 21170.073} C_VEL
LIN {X 0,Y 593.498,Z 1165.446,A -85,B 0,C 180,E1 21167.957,E2 21167.957} C_VEL
LIN {X 0,Y 592.788,Z 1176.303,A -85,B 0,C 180,E1 21165.356,E2 21165.356} C_VEL
LIN {X 0,Y 592.348,Z 1185.178,A -85,B 0,C 180,E1 21162.776,E2 21162.776} C_VEL
LIN {X 0,Y 592.109,Z 1191.859,A -85,B 0,C 180,E1 21160.41,E2 21160.41} C_VEL
LIN {X 0,Y 591.981,Z 1197.541,A -85,B 0,C 180,E1 21157.864,E2 21157.864} C_VEL
LIN {X 0,Y 591.928,Z 1201.66,A -85,B 0,C 180,E1 21155.234,E2 21155.234} C_VEL
LIN {X 0,Y 591.916,Z 1203.924,A -85,B 0,C 180,E1 21152.905,E2 21152.905} C_VEL
LIN {X 0,Y 591.895,Z 1204.849,A -85,B 0,C 180,E1 21150.678,E2 21150.678} C_VEL
LIN {X 0,Y 591.908,Z 1204.623,A -85,B 0,C 180,E1 21148.355,E2 21148.355} C_VEL
LIN {X 0,Y 591.918,Z 1202.789,A -85,B 0,C 180,E1 21145.738,E2 21145.738} C_VEL
LIN {X 0,Y 591.945,Z 1199.546,A -85,B 0,C 180,E1 21143.307,E2 21143.307} C_VEL
LIN {X 0,Y 592.023,Z 1195.103,A -85,B 0,C 180,E1 21140.964,E2 21140.964} C_VEL
LIN {X 0,Y 592.224,Z 1188.472,A -85,B 0,C 180,E1 21138.31,E2 21138.31} C_VEL
LIN {X 0,Y 592.556,Z 1180.572,A -85,B 0,C 180,E1 21135.838,E2 21135.838} C_VEL
LIN {X 0,Y 593.028,Z 1172.305,A -85,B 0,C 180,E1 21133.646,E2 21133.646} C_VEL
LIN {X 0,Y 593.709,Z 1162.694,A -85,B 0,C 180,E1 21131.44,E2 21131.44} C_VEL
LIN {X 0,Y 594.842,Z 1149.447,A -85,B 0,C 180,E1 21128.815,E2 21128.815} C_VEL
LIN {X 0,Y 596.107,Z 1136.315,A -85,B 0,C 180,E1 21126.567,E2 21126.567} C_VEL
LIN {X 0,Y 597.541,Z 1122.985,A -85,B 0,C 180,E1 21124.53,E2 21124.53} C_VEL
LIN {X 0,Y 599.573,Z 1106.412,A -85,B 0,C 180,E1 21122.273,E2 21122.273} C_VEL
LIN {X 0,Y 601.82,Z 1088.228,A -85,B 0,C 180,E1 21120.105,E2 21120.105} C_VEL
LIN {X 0,Y 603.942,Z 1072.289,A -85,B 0,C 180,E1 21118.4,E2 21118.4} C_VEL
LIN {X 0,Y 606.352,Z 1054.611,A -85,B 0,C 180,E1 21116.694,E2 21116.694} C_VEL
LIN {X 0,Y 609.497,Z 1031.563,A -85,B 0,C 180,E1 21114.729,E2 21114.729} C_VEL
LIN {X 0,Y 612.159,Z 1011.513,A -85,B 0,C 180,E1 21113.229,E2 21113.229} C_VEL
LIN {X 0,Y 614.693,Z 992.098,A -85,B 0,C 180,E1 21111.934,E2 21111.934} C_VEL
LIN {X 0,Y 617.675,Z 968.572,A -85,B 0,C 180,E1 21110.549,E2 21110.549} C_VEL
LIN {X 0,Y 620.472,Z 943.978,A -85,B 0,C 180,E1 21109.32,E2 21109.32} C_VEL
LIN {X 0,Y 622.711,Z 922.574,A -85,B 0,C 180,E1 21108.399,E2 21108.399} C_VEL
LIN {X 0,Y 624.664,Z 901.89,A -85,B 0,C 180,E1 21107.633,E2 21107.633} C_VEL
LIN {X 0,Y 626.529,Z 879.591,A -85,B 0,C 180,E1 21106.939,E2 21106.939} C_VEL
LIN {X 0,Y 628.499,Z 850.945,A -85,B 0,C 180,E1 21106.237,E2 21106.237} C_VEL
LIN {X 0,Y 629.695,Z 826.924,A -85,B 0,C 180,E1 21105.806,E2 21105.806} C_VEL
LIN {X 0,Y 633.866,Z 657.273,A -85,B 0,C 180,E1 21103.47,E2 21103.47} C_VEL
LIN {X 0,Y 639.379,Z 440.362,A -85,B 0,C 180,E1 21100.439,E2 21100.439} C_VEL
LIN {X 0,Y 640.065,Z 408.827,A -85,B 0,C 180,E1 21099.974,E2 21099.974} C_VEL
LIN {X 0,Y 626.227,Z 387.878,A -85,B 0,C 180,E1 21098.019,E2 21098.019} C_VEL
LIN {X 0,Y 616.557,Z 374.213,A -85,B 0,C 180,E1 21096.525,E2 21096.525} C_VEL
LIN {X 0,Y 606.8,Z 361.083,A -85,B 0,C 180,E1 21094.904,E2 21094.904} C_VEL
LIN {X 0,Y 603.102,Z 356.144,A -85,B 0,C 180,E1 21094.254,E2 21094.254} C_VEL
LIN {X 0,Y 598.982,Z 351.059,A -85,B 0,C 180,E1 21093.513,E2 21093.513} C_VEL
LIN {X 0,Y 597.022,Z 348.611,A -85,B 0,C 180,E1 21093.092,E2 21093.092} C_VEL
LIN {X 0,Y 595.394,Z 344.937,A -85,B 0,C 180,E1 21092.393,E2 21092.393} C_VEL
LIN {X 0,Y 593.471,Z 341.872,A -85,B 0,C 180,E1 21091.7,E2 21091.7} C_VEL
LIN {X 0,Y 593.107,Z 340.32,A -85,B 0,C 180,E1 21091.395,E2 21091.395} C_VEL
LIN {X 0,Y 593.155,Z 340.346,A -85,B 0,C 180,E1 21088.494,E2 21088.494} C_VEL
LIN {X 0,Y 593.104,Z 340.323,A -85,B 0,C 180,E1 21085.354,E2 21085.354} C_VEL
LIN {X 0,Y 593.13,Z 340.317,A -85,B 0,C 180,E1 21082.5,E2 21082.5} C_VEL
LIN {X 0,Y 593.102,Z 340.352,A -85,B 0,C 180,E1 21079.255,E2 21079.255} C_VEL
LIN {X 0,Y 593.122,Z 340.307,A -85,B 0,C 180,E1 21076.352,E2 21076.352} C_VEL
LIN {X 0,Y 593.1,Z 340.344,A -85,B 0,C 180,E1 21073.155,E2 21073.155} C_VEL
LIN {X 0,Y 593.117,Z 340.317,A -85,B 0,C 180,E1 21070.294,E2 21070.294} C_VEL
LIN {X 0,Y 593.107,Z 340.326,A -85,B 0,C 180,E1 21067.069,E2 21067.069} C_VEL
LIN {X 0,Y 593.116,Z 340.334,A -85,B 0,C 180,E1 21064.254,E2 21064.254} C_VEL
LIN {X 0,Y 593.114,Z 340.311,A -85,B 0,C 180,E1 21060.966,E2 21060.966} C_VEL
LIN {X 0,Y 593.119,Z 340.343,A -85,B 0,C 180,E1 21058.164,E2 21058.164} C_VEL
LIN {X 0,Y 593.122,Z 340.304,A -85,B 0,C 180,E1 21054.874,E2 21054.874} C_VEL
LIN {X 0,Y 593.124,Z 340.349,A -85,B 0,C 180,E1 21052.054,E2 21052.054} C_VEL
LIN {X 0,Y 593.13,Z 340.312,A -85,B 0,C 180,E1 21048.723,E2 21048.723} C_VEL
LIN {X 0,Y 593.132,Z 340.328,A -85,B 0,C 180,E1 21045.851,E2 21045.851} C_VEL
LIN {X 0,Y 593.136,Z 340.339,A -85,B 0,C 180,E1 21042.538,E2 21042.538} C_VEL
LIN {X 0,Y 593.139,Z 340.307,A -85,B 0,C 180,E1 21039.68,E2 21039.68} C_VEL
LIN {X 0,Y 593.136,Z 340.324,A -85,B 0,C 180,E1 21036.346,E2 21036.346} C_VEL
LIN {X 0,Y 593.161,Z 340.504,A -85,B 0,C 180,E1 21033.656,E2 21033.656} C_VEL
LIN {X 0,Y 593.987,Z 342.99,A -85,B 0,C 180,E1 21033.264,E2 21033.264} C_VEL
LIN {X 0,Y 596.375,Z 345.776,A -85,B 0,C 180,E1 21032.814,E2 21032.814} C_VEL
LIN {X 0,Y 597.764,Z 347.289,A -85,B 0,C 180,E1 21032.559,E2 21032.559} C_VEL
LIN {X 0,Y 601.479,Z 351.831,A -85,B 0,C 180,E1 21031.882,E2 21031.882} C_VEL
LIN {X 0,Y 606.81,Z 358.664,A -85,B 0,C 180,E1 21030.943,E2 21030.943} C_VEL
LIN {X 0,Y 611.313,Z 364.427,A -85,B 0,C 180,E1 21030.183,E2 21030.183} C_VEL
LIN {X 0,Y 619.064,Z 374.754,A -85,B 0,C 180,E1 21028.932,E2 21028.932} C_VEL
LIN {X 0,Y 630.698,Z 391.434,A -85,B 0,C 180,E1 21027.18,E2 21027.18} C_VEL
LIN {X 0,Y 640.138,Z 405.789,A -85,B 0,C 180,E1 21025.871,E2 21025.871} C_VEL
LIN {X 0,Y 634.182,Z 636.472,A -85,B 0,C 180,E1 21022.638,E2 21022.638} C_VEL
LIN {X 0,Y 633.986,Z 644.403,A -85,B 0,C 180,E1 21022.528,E2 21022.528} C_VEL
LIN {X 0,Y 633.133,Z 652.103,A -85,B 0,C 180,E1 21022.486,E2 21022.486} C_VEL
LIN {X 0,Y 628.309,Z 672.75,A -85,B 0,C 180,E1 21022.614,E2 21022.614} C_VEL
LIN {X 0,Y 627.601,Z 679.361,A -85,B 0,C 180,E1 21022.574,E2 21022.574} C_VEL
LIN {X 0,Y 623.956,Z 817.569,A -85,B 0,C 180,E1 21020.655,E2 21020.655} C_VEL
LIN {X 0,Y 622.698,Z 841.354,A -85,B 0,C 180,E1 21020.222,E2 21020.222} C_VEL
LIN {X 0,Y 620.624,Z 870.027,A -85,B 0,C 180,E1 21019.516,E2 21019.516} C_VEL
LIN {X 0,Y 618.615,Z 892.797,A -85,B 0,C 180,E1 21018.797,E2 21018.797} C_VEL
LIN {X 0,Y 616.576,Z 913.083,A -85,B 0,C 180,E1 21018.039,E2 21018.039} C_VEL
LIN {X 0,Y 614.333,Z 933.576,A -85,B 0,C 180,E1 21017.15,E2 21017.15} C_VEL
LIN {X 0,Y 611.84,Z 954.462,A -85,B 0,C 180,E1 21016.111,E2 21016.111} C_VEL
LIN {X 0,Y 608.347,Z 981.009,A -85,B 0,C 180,E1 21014.572,E2 21014.572} C_VEL
LIN {X 0,Y 605.606,Z 1000.788,A -85,B 0,C 180,E1 21013.249,E2 21013.249} C_VEL
LIN {X 0,Y 603.015,Z 1019.044,A -85,B 0,C 180,E1 21011.883,E2 21011.883} C_VEL
LIN {X 0,Y 600.179,Z 1039.066,A -85,B 0,C 180,E1 21010.207,E2 21010.207} C_VEL
LIN {X 0,Y 597.083,Z 1060.479,A -85,B 0,C 180,E1 21008.164,E2 21008.164} C_VEL
LIN {X 0,Y 594.75,Z 1076.911,A -85,B 0,C 180,E1 21006.402,E2 21006.402} C_VEL
LIN {X 0,Y 592.598,Z 1092.605,A -85,B 0,C 180,E1 21004.535,E2 21004.535} C_VEL
LIN {X 0,Y 590.308,Z 1110.632,A -85,B 0,C 180,E1 21002.121,E2 21002.121} C_VEL
LIN {X 0,Y 588.607,Z 1124.789,A -85,B 0,C 180,E1 20999.961,E2 20999.961} C_VEL
LIN {X 0,Y 587.319,Z 1136.771,A -85,B 0,C 180,E1 20997.915,E2 20997.915} C_VEL
LIN {X 0,Y 586.138,Z 1149.525,A -85,B 0,C 180,E1 20995.459,E2 20995.459} C_VEL
LIN {X 0,Y 585.197,Z 1161.172,A -85,B 0,C 180,E1 20992.821,E2 20992.821} C_VEL
LIN {X 0,Y 584.678,Z 1169.475,A -85,B 0,C 180,E1 20990.627,E2 20990.627} C_VEL
LIN {X 0,Y 584.297,Z 1176.852,A -85,B 0,C 180,E1 20988.352,E2 20988.352} C_VEL
LIN {X 0,Y 584.079,Z 1183.636,A -85,B 0,C 180,E1 20985.794,E2 20985.794} C_VEL
LIN {X 0,Y 583.961,Z 1188.861,A -85,B 0,C 180,E1 20983.163,E2 20983.163} C_VEL
LIN {X 0,Y 583.921,Z 1192.123,A -85,B 0,C 180,E1 20980.857,E2 20980.857} C_VEL
LIN {X 0,Y 583.915,Z 1194.22,A -85,B 0,C 180,E1 20978.468,E2 20978.468} C_VEL
LIN {X 0,Y 583.895,Z 1194.948,A -85,B 0,C 180,E1 20975.7,E2 20975.7} C_VEL
LIN {X 0,Y 583.911,Z 1194.08,A -85,B 0,C 180,E1 20973.239,E2 20973.239} C_VEL
LIN {X 0,Y 583.924,Z 1192.04,A -85,B 0,C 180,E1 20970.981,E2 20970.981} C_VEL
LIN {X 0,Y 583.966,Z 1188.508,A -85,B 0,C 180,E1 20968.528,E2 20968.528} C_VEL
LIN {X 0,Y 584.099,Z 1182.81,A -85,B 0,C 180,E1 20965.778,E2 20965.778} C_VEL
LIN {X 0,Y 584.346,Z 1176.128,A -85,B 0,C 180,E1 20963.318,E2 20963.318} C_VEL
LIN {X 0,Y 584.728,Z 1168.653,A -85,B 0,C 180,E1 20961.048,E2 20961.048} C_VEL
LIN {X 0,Y 585.399,Z 1158.674,A -85,B 0,C 180,E1 20958.472,E2 20958.472} C_VEL
LIN {X 0,Y 586.368,Z 1146.69,A -85,B 0,C 180,E1 20955.886,E2 20955.886} C_VEL
LIN {X 0,Y 587.491,Z 1135.077,A -85,B 0,C 180,E1 20953.69,E2 20953.69} C_VEL
LIN {X 0,Y 589.186,Z 1120.072,A -85,B 0,C 180,E1 20951.189,E2 20951.189} C_VEL
LIN {X 0,Y 591.081,Z 1104.101,A -85,B 0,C 180,E1 20948.88,E2 20948.88} C_VEL
LIN {X 0,Y 593.045,Z 1089.359,A -85,B 0,C 180,E1 20946.973,E2 20946.973} C_VEL
LIN {X 0,Y 595.581,Z 1071.205,A -85,B 0,C 180,E1 20944.865,E2 20944.865} C_VEL
LIN {X 0,Y 598.428,Z 1050.965,A -85,B 0,C 180,E1 20942.808,E2 20942.808} C_VEL
LIN {X 0,Y 600.879,Z 1033.903,A -85,B 0,C 180,E1 20941.255,E2 20941.255} C_VEL
LIN {X 0,Y 603.426,Z 1016.244,A -85,B 0,C 180,E1 20939.808,E2 20939.808} C_VEL
LIN {X 0,Y 606.667,Z 993.82,A -85,B 0,C 180,E1 20938.169,E2 20938.169} C_VEL
LIN {X 0,Y 609.819,Z 970.175,A -85,B 0,C 180,E1 20936.682,E2 20936.682} C_VEL
LIN {X 0,Y 612.2,Z 951.506,A -85,B 0,C 180,E1 20935.647,E2 20935.647} C_VEL
LIN {X 0,Y 614.454,Z 932.527,A -85,B 0,C 180,E1 20934.712,E2 20934.712} C_VEL
LIN {X 0,Y 616.685,Z 912.066,A -85,B 0,C 180,E1 20933.83,E2 20933.83} C_VEL
LIN {X 0,Y 618.791,Z 891.018,A -85,B 0,C 180,E1 20933.051,E2 20933.051} C_VEL
LIN {X 0,Y 621.12,Z 864.471,A -85,B 0,C 180,E1 20932.239,E2 20932.239} C_VEL
LIN {X 0,Y 622.83,Z 838.863,A -85,B 0,C 180,E1 20931.638,E2 20931.638} C_VEL
LIN {X 0,Y 623.998,Z 816.482,A -85,B 0,C 180,E1 20931.238,E2 20931.238} C_VEL
LIN {X 0,Y 629.357,Z 611.541,A -85,B 0,C 180,E1 20928.392,E2 20928.392} C_VEL
LIN {X 0,Y 634.836,Z 409.462,A -85,B 0,C 180,E1 20925.53,E2 20925.53} C_VEL
LIN {X 0,Y 621.542,Z 390.241,A -85,B 0,C 180,E1 20923.706,E2 20923.706} C_VEL
LIN {X 0,Y 607.632,Z 371.427,A -85,B 0,C 180,E1 20921.699,E2 20921.699} C_VEL
LIN {X 0,Y 597.522,Z 357.99,A -85,B 0,C 180,E1 20920.142,E2 20920.142} C_VEL
LIN {X 0,Y 593.082,Z 352.479,A -85,B 0,C 180,E1 20919.433,E2 20919.433} C_VEL
LIN {X 0,Y 590.363,Z 348.938,A -85,B 0,C 180,E1 20918.985,E2 20918.985} C_VEL
LIN {X 0,Y 589.125,Z 347.233,A -85,B 0,C 180,E1 20918.777,E2 20918.777} C_VEL
LIN {X 0,Y 586.483,Z 344.739,A -85,B 0,C 180,E1 20918.349,E2 20918.349} C_VEL
LIN {X 0,Y 585.31,Z 341.86,A -85,B 0,C 180,E1 20918.076,E2 20918.076} C_VEL
LIN {X 0,Y 585.229,Z 341.328,A -85,B 0,C 180,E1 20917.958,E2 20917.958} C_VEL
LIN {X 0,Y 585.249,Z 341.331,A -85,B 0,C 180,E1 20914.676,E2 20914.676} C_VEL
LIN {X 0,Y 585.256,Z 341.328,A -85,B 0,C 180,E1 20911.405,E2 20911.405} C_VEL
LIN {X 0,Y 585.217,Z 341.314,A -85,B 0,C 180,E1 20908.136,E2 20908.136} C_VEL
LIN {X 0,Y 585.257,Z 341.3,A -85,B 0,C 180,E1 20904.96,E2 20904.96} C_VEL
LIN {X 0,Y 585.206,Z 341.306,A -85,B 0,C 180,E1 20901.869,E2 20901.869} C_VEL
LIN {X 0,Y 585.256,Z 341.302,A -85,B 0,C 180,E1 20898.632,E2 20898.632} C_VEL
LIN {X 0,Y 585.202,Z 341.312,A -85,B 0,C 180,E1 20895.56,E2 20895.56} C_VEL
LIN {X 0,Y 585.237,Z 341.291,A -85,B 0,C 180,E1 20892.331,E2 20892.331} C_VEL
LIN {X 0,Y 585.199,Z 341.329,A -85,B 0,C 180,E1 20889.342,E2 20889.342} C_VEL
LIN {X 0,Y 585.223,Z 341.326,A -85,B 0,C 180,E1 20886.081,E2 20886.081} C_VEL
LIN {X 0,Y 585.202,Z 341.334,A -85,B 0,C 180,E1 20883.036,E2 20883.036} C_VEL
LIN {X 0,Y 585.195,Z 341.335,A -85,B 0,C 180,E1 20879.706,E2 20879.706} C_VEL
LIN {X 0,Y 585.204,Z 341.331,A -85,B 0,C 180,E1 20876.768,E2 20876.768} C_VEL
LIN {X 0,Y 585.185,Z 341.338,A -85,B 0,C 180,E1 20873.525,E2 20873.525} C_VEL
LIN {X 0,Y 585.193,Z 341.325,A -85,B 0,C 180,E1 20870.658,E2 20870.658} C_VEL
LIN {X 0,Y 585.17,Z 341.296,A -85,B 0,C 180,E1 20867.366,E2 20867.366} C_VEL
LIN {X 0,Y 585.187,Z 341.321,A -85,B 0,C 180,E1 20864.51,E2 20864.51} C_VEL
LIN {X 0,Y 585.165,Z 341.298,A -85,B 0,C 180,E1 20861.262,E2 20861.262} C_VEL
LIN {X 0,Y 585.183,Z 341.327,A -85,B 0,C 180,E1 20858.341,E2 20858.341} C_VEL
LIN {X 0,Y 585.16,Z 341.29,A -85,B 0,C 180,E1 20855.14,E2 20855.14} C_VEL
LIN {X 0,Y 585.189,Z 341.339,A -85,B 0,C 180,E1 20852.195,E2 20852.195} C_VEL
LIN {X 0,Y 585.169,Z 341.33,A -85,B 0,C 180,E1 20848.933,E2 20848.933} C_VEL
LIN {X 0,Y 585.194,Z 341.557,A -85,B 0,C 180,E1 20848.706,E2 20848.706} C_VEL
LIN {X 0,Y 586.649,Z 345.028,A -85,B 0,C 180,E1 20848.105,E2 20848.105} C_VEL
LIN {X 0,Y 587.663,Z 346.28,A -85,B 0,C 180,E1 20847.821,E2 20847.821} C_VEL
LIN {X 0,Y 589.253,Z 349.814,A -85,B 0,C 180,E1 20847.256,E2 20847.256} C_VEL
LIN {X 0,Y 594.36,Z 356.171,A -85,B 0,C 180,E1 20846.423,E2 20846.423} C_VEL
LIN {X 0,Y 610.364,Z 377.935,A -85,B 0,C 180,E1 20843.948,E2 20843.948} C_VEL
LIN {X 0,Y 624.523,Z 397.559,A -85,B 0,C 180,E1 20841.931,E2 20841.931} C_VEL
LIN {X 0,Y 634.932,Z 413.065,A -85,B 0,C 180,E1 20840.507,E2 20840.507} C_VEL
LIN {X 0,Y 629.42,Z 616.476,A -85,B 0,C 180,E1 20837.629,E2 20837.629} C_VEL
LIN {X 0,Y 624.018,Z 825.223,A -85,B 0,C 180,E1 20834.733,E2 20834.733} C_VEL
LIN {X 0,Y 622.887,Z 847.314,A -85,B 0,C 180,E1 20834.345,E2 20834.345} C_VEL
LIN {X 0,Y 621.248,Z 872.195,A -85,B 0,C 180,E1 20833.772,E2 20833.772} C_VEL
LIN {X 0,Y 618.935,Z 899.295,A -85,B 0,C 180,E1 20832.96,E2 20832.96} C_VEL
LIN {X 0,Y 616.844,Z 920.613,A -85,B 0,C 180,E1 20832.182,E2 20832.182} C_VEL
LIN {X 0,Y 614.686,Z 940.562,A -85,B 0,C 180,E1 20831.332,E2 20831.332} C_VEL
LIN {X 0,Y 612.545,Z 958.662,A -85,B 0,C 180,E1 20830.455,E2 20830.455} C_VEL
LIN {X 0,Y 610.14,Z 977.615,A -85,B 0,C 180,E1 20829.422,E2 20829.422} C_VEL
LIN {X 0,Y 607.447,Z 997.852,A -85,B 0,C 180,E1 20828.177,E2 20828.177} C_VEL
LIN {X 0,Y 603.999,Z 1022.551,A -85,B 0,C 180,E1 20826.433,E2 20826.433} C_VEL
LIN {X 0,Y 601.135,Z 1042.213,A -85,B 0,C 180,E1 20824.845,E2 20824.845} C_VEL
LIN {X 0,Y 598.622,Z 1059.597,A -85,B 0,C 180,E1 20823.278,E2 20823.278} C_VEL
LIN {X 0,Y 595.845,Z 1079.323,A -85,B 0,C 180,E1 20821.296,E2 20821.296} C_VEL
LIN {X 0,Y 593.242,Z 1097.983,A -85,B 0,C 180,E1 20819.15,E2 20819.15} C_VEL
LIN {X 0,Y 591.278,Z 1112.608,A -85,B 0,C 180,E1 20817.276,E2 20817.276} C_VEL
LIN {X 0,Y 589.497,Z 1127.18,A -85,B 0,C 180,E1 20815.197,E2 20815.197} C_VEL
LIN {X 0,Y 587.644,Z 1143.701,A -85,B 0,C 180,E1 20812.51,E2 20812.51} C_VEL
LIN {X 0,Y 586.478,Z 1155.375,A -85,B 0,C 180,E1 20810.331,E2 20810.331} C_VEL
LIN {X 0,Y 585.631,Z 1165.444,A -85,B 0,C 180,E1 20808.207,E2 20808.207} C_VEL
LIN {X 0,Y 584.858,Z 1176.305,A -85,B 0,C 180,E1 20805.57,E2 20805.57} C_VEL
LIN {X 0,Y 584.389,Z 1185.175,A -85,B 0,C 180,E1 20802.953,E2 20802.953} C_VEL
LIN {X 0,Y 584.129,Z 1191.602,A -85,B 0,C 180,E1 20800.654,E2 20800.654} C_VEL
LIN {X 0,Y 583.992,Z 1197.15,A -85,B 0,C 180,E1 20798.17,E2 20798.17} C_VEL
LIN {X 0,Y 583.929,Z 1201.427,A -85,B 0,C 180,E1 20795.503,E2 20795.503} C_VEL
LIN {X 0,Y 583.917,Z 1203.854,A -85,B 0,C 180,E1 20793.043,E2 20793.043} C_VEL
LIN {X 0,Y 583.905,Z 1204.804,A -85,B 0,C 180,E1 20790.883,E2 20790.883} C_VEL
LIN {X 0,Y 583.915,Z 1204.736,A -85,B 0,C 180,E1 20788.823,E2 20788.823} C_VEL
LIN {X 0,Y 583.913,Z 1203.51,A -85,B 0,C 180,E1 20786.466,E2 20786.466} C_VEL
LIN {X 0,Y 583.943,Z 1200.337,A -85,B 0,C 180,E1 20783.709,E2 20783.709} C_VEL
LIN {X 0,Y 584.019,Z 1195.926,A -85,B 0,C 180,E1 20781.236,E2 20781.236} C_VEL
LIN {X 0,Y 584.152,Z 1190.586,A -85,B 0,C 180,E1 20778.948,E2 20778.948} C_VEL
LIN {X 0,Y 584.519,Z 1182.686,A -85,B 0,C 180,E1 20776.245,E2 20776.245} C_VEL
LIN {X 0,Y 585.07,Z 1173.114,A -85,B 0,C 180,E1 20773.622,E2 20773.622} C_VEL
LIN {X 0,Y 585.744,Z 1164.075,A -85,B 0,C 180,E1 20771.488,E2 20771.488} C_VEL
LIN {X 0,Y 586.693,Z 1153.206,A -85,B 0,C 180,E1 20769.239,E2 20769.239} C_VEL
LIN {X 0,Y 588.226,Z 1138.277,A -85,B 0,C 180,E1 20766.562,E2 20766.562} C_VEL
LIN {X 0,Y 589.783,Z 1124.559,A -85,B 0,C 180,E1 20764.413,E2 20764.413} C_VEL
LIN {X 0,Y 591.601,Z 1110.302,A -85,B 0,C 180,E1 20762.414,E2 20762.414} C_VEL
LIN {X 0,Y 594.107,Z 1091.613,A -85,B 0,C 180,E1 20760.084,E2 20760.084} C_VEL
LIN {X 0,Y 596.593,Z 1073.808,A -85,B 0,C 180,E1 20758.135,E2 20758.135} C_VEL
LIN {X 0,Y 598.948,Z 1057.385,A -85,B 0,C 180,E1 20756.515,E2 20756.515} C_VEL
LIN {X 0,Y 601.696,Z 1038.575,A -85,B 0,C 180,E1 20754.846,E2 20754.846} C_VEL
LIN {X 0,Y 605.029,Z 1015.184,A -85,B 0,C 180,E1 20753.02,E2 20753.02} C_VEL
LIN {X 0,Y 607.751,Z 995.422,A -85,B 0,C 180,E1 20751.667,E2 20751.667} C_VEL
LIN {X 0,Y 610.362,Z 975.83,A -85,B 0,C 180,E1 20750.475,E2 20750.475} C_VEL
LIN {X 0,Y 612.907,Z 955.669,A -85,B 0,C 180,E1 20749.39,E2 20749.39} C_VEL
LIN {X 0,Y 615.756,Z 931.531,A -85,B 0,C 180,E1 20748.26,E2 20748.26} C_VEL
LIN {X 0,Y 618.273,Z 906.28,A -85,B 0,C 180,E1 20747.28,E2 20747.28} C_VEL
LIN {X 0,Y 620.184,Z 884.886,A -85,B 0,C 180,E1 20746.587,E2 20746.587} C_VEL
LIN {X 0,Y 621.82,Z 863.659,A -85,B 0,C 180,E1 20746.017,E2 20746.017} C_VEL
LIN {X 0,Y 623.18,Z 842.094,A -85,B 0,C 180,E1 20745.553,E2 20745.553} C_VEL
LIN {X 0,Y 624.439,Z 814.38,A -85,B 0,C 180,E1 20745.105,E2 20745.105} C_VEL
LIN {X 0,Y 630.053,Z 592.045,A -85,B 0,C 180,E1 20742.03,E2 20742.03} C_VEL
LIN {X 0,Y 634.917,Z 412.86,A -85,B 0,C 180,E1 20739.485,E2 20739.485} C_VEL
LIN {X 0,Y 620.822,Z 391.464,A -85,B 0,C 180,E1 20737.416,E2 20737.416} C_VEL
LIN {X 0,Y 610.738,Z 377.075,A -85,B 0,C 180,E1 20735.795,E2 20735.795} C_VEL
LIN {X 0,Y 603.071,Z 367.052,A -85,B 0,C 180,E1 20734.486,E2 20734.486} C_VEL
LIN {X 0,Y 598.833,Z 361.503,A -85,B 0,C 180,E1 20733.724,E2 20733.724} C_VEL
LIN {X 0,Y 594.455,Z 355.957,A -85,B 0,C 180,E1 20732.908,E2 20732.908} C_VEL
LIN {X 0,Y 590.071,Z 350.529,A -85,B 0,C 180,E1 20732.06,E2 20732.06} C_VEL
LIN {X 0,Y 588.48,Z 348.343,A -85,B 0,C 180,E1 20731.67,E2 20731.67} C_VEL
LIN {X 0,Y 587.678,Z 346.197,A -85,B 0,C 180,E1 20731.261,E2 20731.261} C_VEL
LIN {X 0,Y 585.792,Z 343.45,A -85,B 0,C 180,E1 20730.575,E2 20730.575} C_VEL
LIN {X 0,Y 585.235,Z 341.294,A -85,B 0,C 180,E1 20730.153,E2 20730.153} C_VEL
LIN {X 0,Y 585.163,Z 341.307,A -85,B 0,C 180,E1 20727.144,E2 20727.144} C_VEL
LIN {X 0,Y 585.229,Z 341.336,A -85,B 0,C 180,E1 20723.994,E2 20723.994} C_VEL
LIN {X 0,Y 585.154,Z 341.303,A -85,B 0,C 180,E1 20721.029,E2 20721.029} C_VEL
LIN {X 0,Y 585.225,Z 341.308,A -85,B 0,C 180,E1 20717.911,E2 20717.911} C_VEL
LIN {X 0,Y 585.152,Z 341.33,A -85,B 0,C 180,E1 20714.852,E2 20714.852} C_VEL
LIN {X 0,Y 585.224,Z 341.29,A -85,B 0,C 180,E1 20711.768,E2 20711.768} C_VEL
LIN {X 0,Y 585.156,Z 341.34,A -85,B 0,C 180,E1 20708.747,E2 20708.747} C_VEL
LIN {X 0,Y 585.235,Z 341.287,A -85,B 0,C 180,E1 20705.687,E2 20705.687} C_VEL
LIN {X 0,Y 585.165,Z 341.338,A -85,B 0,C 180,E1 20702.644,E2 20702.644} C_VEL
LIN {X 0,Y 585.245,Z 341.29,A -85,B 0,C 180,E1 20699.511,E2 20699.511} C_VEL
LIN {X 0,Y 585.168,Z 341.325,A -85,B 0,C 180,E1 20696.473,E2 20696.473} C_VEL
LIN {X 0,Y 585.25,Z 341.305,A -85,B 0,C 180,E1 20693.328,E2 20693.328} C_VEL
LIN {X 0,Y 585.173,Z 341.303,A -85,B 0,C 180,E1 20690.261,E2 20690.261} C_VEL
LIN {X 0,Y 585.24,Z 341.333,A -85,B 0,C 180,E1 20687.067,E2 20687.067} C_VEL
LIN {X 0,Y 585.178,Z 341.292,A -85,B 0,C 180,E1 20684.134,E2 20684.134} C_VEL
LIN {X 0,Y 585.244,Z 341.309,A -85,B 0,C 180,E1 20680.954,E2 20680.954} C_VEL
LIN {X 0,Y 585.189,Z 341.328,A -85,B 0,C 180,E1 20677.92,E2 20677.92} C_VEL
LIN {X 0,Y 585.258,Z 341.324,A -85,B 0,C 180,E1 20674.932,E2 20674.932} C_VEL
LIN {X 0,Y 585.743,Z 343.28,A -85,B 0,C 180,E1 20674.656,E2 20674.656} C_VEL
LIN {X 0,Y 587.629,Z 346.123,A -85,B 0,C 180,E1 20674.257,E2 20674.257} C_VEL
LIN {X 0,Y 590.135,Z 348.176,A -85,B 0,C 180,E1 20673.781,E2 20673.781} C_VEL
LIN {X 0,Y 593.206,Z 352.41,A -85,B 0,C 180,E1 20673.172,E2 20673.172} C_VEL
LIN {X 0,Y 595.165,Z 354.458,A -85,B 0,C 180,E1 20672.808,E2 20672.808} C_VEL
LIN {X 0,Y 603.656,Z 365.183,A -85,B 0,C 180,E1 20671.264,E2 20671.264} C_VEL
LIN {X 0,Y 611.414,Z 375.309,A -85,B 0,C 180,E1 20669.945,E2 20669.945} C_VEL
LIN {X 0,Y 620.902,Z 388.586,A -85,B 0,C 180,E1 20668.427,E2 20668.427} C_VEL
LIN {X 0,Y 634.228,Z 408.492,A -85,B 0,C 180,E1 20666.469,E2 20666.469} C_VEL
LIN {X 0,Y 634.895,Z 409.865,A -85,B 0,C 180,E1 20666.37,E2 20666.37} C_VEL
LIN {X 0,Y 628.656,Z 638.157,A -85,B 0,C 180,E1 20663.148,E2 20663.148} C_VEL
LIN {X 0,Y 627.601,Z 679.361,A -85,B 0,C 180,E1 20662.574,E2 20662.574} C_VEL
LIN {X 0,Y 626.691,Z 687.067,A -85,B 0,C 180,E1 20662.536,E2 20662.536} C_VEL
LIN {X 0,Y 621.838,Z 707.703,A -85,B 0,C 180,E1 20662.669,E2 20662.669} C_VEL
LIN {X 0,Y 621.162,Z 714.308,A -85,B 0,C 180,E1 20662.626,E2 20662.626} C_VEL
LIN {X 0,Y 618.248,Z 818.246,A -85,B 0,C 180,E1 20661.168,E2 20661.168} C_VEL
LIN {X 0,Y 616.785,Z 844.492,A -85,B 0,C 180,E1 20660.681,E2 20660.681} C_VEL
LIN {X 0,Y 614.623,Z 871.959,A -85,B 0,C 180,E1 20659.979,E2 20659.979} C_VEL
LIN {X 0,Y 612.646,Z 893.357,A -85,B 0,C 180,E1 20659.296,E2 20659.296} C_VEL
LIN {X 0,Y 610.423,Z 914.38,A -85,B 0,C 180,E1 20658.501,E2 20658.501} C_VEL
LIN {X 0,Y 607.741,Z 937.417,A -85,B 0,C 180,E1 20657.481,E2 20657.481} C_VEL
LIN {X 0,Y 604.325,Z 963.568,A -85,B 0,C 180,E1 20656.111,E2 20656.111} C_VEL
LIN {X 0,Y 601.49,Z 983.818,A -85,B 0,C 180,E1 20654.882,E2 20654.882} C_VEL
LIN {X 0,Y 598.753,Z 1002.551,A -85,B 0,C 180,E1 20653.604,E2 20653.604} C_VEL
LIN {X 0,Y 595.726,Z 1022.945,A -85,B 0,C 180,E1 20652.042,E2 20652.042} C_VEL
LIN {X 0,Y 592.388,Z 1044.871,A -85,B 0,C 180,E1 20650.127,E2 20650.127} C_VEL
LIN {X 0,Y 589.756,Z 1062.028,A -85,B 0,C 180,E1 20648.437,E2 20648.437} C_VEL
LIN {X 0,Y 587.364,Z 1078.006,A -85,B 0,C 180,E1 20646.691,E2 20646.691} C_VEL
LIN {X 0,Y 584.867,Z 1095.375,A -85,B 0,C 180,E1 20644.581,E2 20644.581} C_VEL
LIN {X 0,Y 582.475,Z 1112.879,A -85,B 0,C 180,E1 20642.15,E2 20642.15} C_VEL
LIN {X 0,Y 580.796,Z 1126.198,A -85,B 0,C 180,E1 20640.064,E2 20640.064} C_VEL
LIN {X 0,Y 579.282,Z 1139.83,A -85,B 0,C 180,E1 20637.665,E2 20637.665} C_VEL
LIN {X 0,Y 577.98,Z 1153.018,A -85,B 0,C 180,E1 20634.967,E2 20634.967} C_VEL
LIN {X 0,Y 577.212,Z 1162.486,A -85,B 0,C 180,E1 20632.723,E2 20632.723} C_VEL
LIN {X 0,Y 576.671,Z 1170.618,A -85,B 0,C 180,E1 20630.502,E2 20630.502} C_VEL
LIN {X 0,Y 576.274,Z 1178.72,A -85,B 0,C 180,E1 20627.885,E2 20627.885} C_VEL
LIN {X 0,Y 576.043,Z 1185.23,A -85,B 0,C 180,E1 20625.18,E2 20625.18} C_VEL
LIN {X 0,Y 575.951,Z 1189.533,A -85,B 0,C 180,E1 20622.839,E2 20622.839} C_VEL
LIN {X 0,Y 575.919,Z 1192.714,A -85,B 0,C 180,E1 20620.402,E2 20620.402} C_VEL
LIN {X 0,Y 575.907,Z 1194.615,A -85,B 0,C 180,E1 20617.682,E2 20617.682} C_VEL
LIN {X 0,Y 575.902,Z 1194.854,A -85,B 0,C 180,E1 20615.279,E2 20615.279} C_VEL
LIN {X 0,Y 575.913,Z 1193.998,A -85,B 0,C 180,E1 20613.085,E2 20613.085} C_VEL
LIN {X 0,Y 575.925,Z 1191.906,A -85,B 0,C 180,E1 20610.795,E2 20610.795} C_VEL
LIN {X 0,Y 575.97,Z 1188.313,A -85,B 0,C 180,E1 20608.308,E2 20608.308} C_VEL
LIN {X 0,Y 576.12,Z 1182.523,A -85,B 0,C 180,E1 20605.52,E2 20605.52} C_VEL
LIN {X 0,Y 576.386,Z 1176.079,A -85,B 0,C 180,E1 20603.125,E2 20603.125} C_VEL
LIN {X 0,Y 576.792,Z 1168.601,A -85,B 0,C 180,E1 20600.823,E2 20600.823} C_VEL
LIN {X 0,Y 577.534,Z 1158.618,A -85,B 0,C 180,E1 20598.212,E2 20598.212} C_VEL
LIN {X 0,Y 578.568,Z 1146.62,A -85,B 0,C 180,E1 20595.59,E2 20595.59} C_VEL
LIN {X 0,Y 579.713,Z 1135.555,A -85,B 0,C 180,E1 20593.465,E2 20593.465} C_VEL
LIN {X 0,Y 581.406,Z 1121.439,A -85,B 0,C 180,E1 20591.065,E2 20591.065} C_VEL
LIN {X 0,Y 583.532,Z 1104.744,A -85,B 0,C 180,E1 20588.594,E2 20588.594} C_VEL
LIN {X 0,Y 585.613,Z 1090.063,A -85,B 0,C 180,E1 20586.664,E2 20586.664} C_VEL
LIN {X 0,Y 588,Z 1073.769,A -85,B 0,C 180,E1 20584.734,E2 20584.734} C_VEL
LIN {X 0,Y 591.214,Z 1052.417,A -85,B 0,C 180,E1 20582.503,E2 20582.503} C_VEL
LIN {X 0,Y 593.955,Z 1034.39,A -85,B 0,C 180,E1 20580.839,E2 20580.839} C_VEL
LIN {X 0,Y 596.653,Z 1016.706,A -85,B 0,C 180,E1 20579.373,E2 20579.373} C_VEL
LIN {X 0,Y 599.712,Z 996.422,A -85,B 0,C 180,E1 20577.869,E2 20577.869} C_VEL
LIN {X 0,Y 603.255,Z 971.636,A -85,B 0,C 180,E1 20576.272,E2 20576.272} C_VEL
LIN {X 0,Y 605.988,Z 951.225,A -85,B 0,C 180,E1 20575.129,E2 20575.129} C_VEL
LIN {X 0,Y 608.373,Z 932.226,A -85,B 0,C 180,E1 20574.19,E2 20574.19} C_VEL
LIN {X 0,Y 610.712,Z 911.748,A -85,B 0,C 180,E1 20573.302,E2 20573.302} C_VEL
LIN {X 0,Y 613.077,Z 889.234,A -85,B 0,C 180,E1 20572.472,E2 20572.472} C_VEL
LIN {X 0,Y 615.543,Z 861.066,A -85,B 0,C 180,E1 20571.631,E2 20571.631} C_VEL
LIN {X 0,Y 617.173,Z 837.652,A -85,B 0,C 180,E1 20571.09,E2 20571.09} C_VEL
LIN {X 0,Y 618.384,Z 815.059,A -85,B 0,C 180,E1 20570.692,E2 20570.692} C_VEL
LIN {X 0,Y 624.263,Z 600.677,A -85,B 0,C 180,E1 20567.694,E2 20567.694} C_VEL
LIN {X 0,Y 629.579,Z 413.37,A -85,B 0,C 180,E1 20565.021,E2 20565.021} C_VEL
LIN {X 0,Y 614.667,Z 391.98,A -85,B 0,C 180,E1 20562.937,E2 20562.937} C_VEL
LIN {X 0,Y 599.629,Z 371.799,A -85,B 0,C 180,E1 20560.693,E2 20560.693} C_VEL
LIN {X 0,Y 593.727,Z 364.035,A -85,B 0,C 180,E1 20559.757,E2 20559.757} C_VEL
LIN {X 0,Y 589.846,Z 359.143,A -85,B 0,C 180,E1 20559.126,E2 20559.126} C_VEL
LIN {X 0,Y 586.69,Z 354.785,A -85,B 0,C 180,E1 20558.592,E2 20558.592} C_VEL
LIN {X 0,Y 583.223,Z 351.217,A -85,B 0,C 180,E1 20558.018,E2 20558.018} C_VEL
LIN {X 0,Y 581.672,Z 348.484,A -85,B 0,C 180,E1 20557.732,E2 20557.732} C_VEL
LIN {X 0,Y 578.858,Z 346.124,A -85,B 0,C 180,E1 20557.261,E2 20557.261} C_VEL
LIN {X 0,Y 577.468,Z 343.153,A -85,B 0,C 180,E1 20556.984,E2 20556.984} C_VEL
LIN {X 0,Y 577.319,Z 342.319,A -85,B 0,C 180,E1 20556.919,E2 20556.919} C_VEL
LIN {X 0,Y 577.299,Z 342.315,A -85,B 0,C 180,E1 20553.659,E2 20553.659} C_VEL
LIN {X 0,Y 577.291,Z 342.312,A -85,B 0,C 180,E1 20550.382,E2 20550.382} C_VEL
LIN {X 0,Y 577.313,Z 342.27,A -85,B 0,C 180,E1 20547.209,E2 20547.209} C_VEL
LIN {X 0,Y 577.274,Z 342.323,A -85,B 0,C 180,E1 20543.911,E2 20543.911} C_VEL
LIN {X 0,Y 577.319,Z 342.261,A -85,B 0,C 180,E1 20540.732,E2 20540.732} C_VEL
LIN {X 0,Y 577.271,Z 342.321,A -85,B 0,C 180,E1 20537.541,E2 20537.541} C_VEL
LIN {X 0,Y 577.284,Z 342.261,A -85,B 0,C 180,E1 20534.238,E2 20534.238} C_VEL
LIN {X 0,Y 577.274,Z 342.315,A -85,B 0,C 180,E1 20531.186,E2 20531.186} C_VEL
LIN {X 0,Y 577.264,Z 342.317,A -85,B 0,C 180,E1 20527.865,E2 20527.865} C_VEL
LIN {X 0,Y 577.281,Z 342.307,A -85,B 0,C 180,E1 20524.869,E2 20524.869} C_VEL
LIN {X 0,Y 577.249,Z 342.311,A -85,B 0,C 180,E1 20521.588,E2 20521.588} C_VEL
LIN {X 0,Y 577.291,Z 342.312,A -85,B 0,C 180,E1 20518.611,E2 20518.611} C_VEL
LIN {X 0,Y 577.242,Z 342.319,A -85,B 0,C 180,E1 20515.43,E2 20515.43} C_VEL
LIN {X 0,Y 577.302,Z 342.317,A -85,B 0,C 180,E1 20512.336,E2 20512.336} C_VEL
LIN {X 0,Y 577.232,Z 342.326,A -85,B 0,C 180,E1 20509.16,E2 20509.16} C_VEL
LIN {X 0,Y 577.296,Z 342.264,A -85,B 0,C 180,E1 20505.967,E2 20505.967} C_VEL
LIN {X 0,Y 577.225,Z 342.328,A -85,B 0,C 180,E1 20502.874,E2 20502.874} C_VEL
LIN {X 0,Y 577.273,Z 342.272,A -85,B 0,C 180,E1 20499.731,E2 20499.731} C_VEL
LIN {X 0,Y 577.216,Z 342.323,A -85,B 0,C 180,E1 20496.845,E2 20496.845} C_VEL
LIN {X 0,Y 577.283,Z 342.28,A -85,B 0,C 180,E1 20493.678,E2 20493.678} C_VEL
LIN {X 0,Y 577.223,Z 342.321,A -85,B 0,C 180,E1 20490.611,E2 20490.611} C_VEL
LIN {X 0,Y 577.303,Z 342.37,A -85,B 0,C 180,E1 20489.798,E2 20489.798} C_VEL
LIN {X 0,Y 578.603,Z 345.875,A -85,B 0,C 180,E1 20489.189,E2 20489.189} C_VEL
LIN {X 0,Y 579.798,Z 347.696,A -85,B 0,C 180,E1 20488.8,E2 20488.8} C_VEL
LIN {X 0,Y 580.805,Z 349.863,A -85,B 0,C 180,E1 20488.471,E2 20488.471} C_VEL
LIN {X 0,Y 584.265,Z 354.174,A -85,B 0,C 180,E1 20487.872,E2 20487.872} C_VEL
LIN {X 0,Y 592.455,Z 364.845,A -85,B 0,C 180,E1 20486.504,E2 20486.504} C_VEL
LIN {X 0,Y 603.908,Z 380.29,A -85,B 0,C 180,E1 20484.701,E2 20484.701} C_VEL
LIN {X 0,Y 619.76,Z 402.216,A -85,B 0,C 180,E1 20482.389,E2 20482.389} C_VEL
LIN {X 0,Y 629.689,Z 417.108,A -85,B 0,C 180,E1 20481.01,E2 20481.01} C_VEL
LIN {X 0,Y 623.898,Z 620.961,A -85,B 0,C 180,E1 20478.11,E2 20478.11} C_VEL
LIN {X 0,Y 618.294,Z 825.921,A -85,B 0,C 180,E1 20475.244,E2 20475.244} C_VEL
LIN {X 0,Y 617.064,Z 848.634,A -85,B 0,C 180,E1 20474.839,E2 20474.839} C_VEL
LIN {X 0,Y 615.089,Z 876.263,A -85,B 0,C 180,E1 20474.18,E2 20474.18} C_VEL
LIN {X 0,Y 612.931,Z 899.924,A -85,B 0,C 180,E1 20473.453,E2 20473.453} C_VEL
LIN {X 0,Y 610.742,Z 921.154,A -85,B 0,C 180,E1 20472.671,E2 20472.671} C_VEL
LIN {X 0,Y 608.562,Z 940.511,A -85,B 0,C 180,E1 20471.841,E2 20471.841} C_VEL
LIN {X 0,Y 606.27,Z 958.977,A -85,B 0,C 180,E1 20470.943,E2 20470.943} C_VEL
LIN {X 0,Y 603.663,Z 978.512,A -85,B 0,C 180,E1 20469.867,E2 20469.867} C_VEL
LIN {X 0,Y 600.521,Z 1001.095,A -85,B 0,C 180,E1 20468.454,E2 20468.454} C_VEL
LIN {X 0,Y 597.053,Z 1024.21,A -85,B 0,C 180,E1 20466.777,E2 20466.777} C_VEL
LIN {X 0,Y 594.205,Z 1042.819,A -85,B 0,C 180,E1 20465.252,E2 20465.252} C_VEL
LIN {X 0,Y 591.553,Z 1060.151,A -85,B 0,C 180,E1 20463.67,E2 20463.67} C_VEL
LIN {X 0,Y 588.527,Z 1080.334,A -85,B 0,C 180,E1 20461.61,E2 20461.61} C_VEL
LIN {X 0,Y 585.85,Z 1098.46,A -85,B 0,C 180,E1 20459.49,E2 20459.49} C_VEL
LIN {X 0,Y 583.725,Z 1113.376,A -85,B 0,C 180,E1 20457.548,E2 20457.548} C_VEL
LIN {X 0,Y 581.68,Z 1129.279,A -85,B 0,C 180,E1 20455.233,E2 20455.233} C_VEL
LIN {X 0,Y 579.853,Z 1144.403,A -85,B 0,C 180,E1 20452.698,E2 20452.698} C_VEL
LIN {X 0,Y 578.642,Z 1155.778,A -85,B 0,C 180,E1 20450.535,E2 20450.535} C_VEL
LIN {X 0,Y 577.698,Z 1166.36,A -85,B 0,C 180,E1 20448.257,E2 20448.257} C_VEL
LIN {X 0,Y 576.866,Z 1177.388,A -85,B 0,C 180,E1 20445.479,E2 20445.479} C_VEL
LIN {X 0,Y 576.433,Z 1185.172,A -85,B 0,C 180,E1 20443.134,E2 20443.134} C_VEL
LIN {X 0,Y 576.142,Z 1191.611,A -85,B 0,C 180,E1 20440.798,E2 20440.798} C_VEL
LIN {X 0,Y 575.999,Z 1197.15,A -85,B 0,C 180,E1 20438.284,E2 20438.284} C_VEL
LIN {X 0,Y 575.93,Z 1201.427,A -85,B 0,C 180,E1 20435.58,E2 20435.58} C_VEL
LIN {X 0,Y 575.917,Z 1203.851,A -85,B 0,C 180,E1 20433.086,E2 20433.086} C_VEL
LIN {X 0,Y 575.905,Z 1204.804,A -85,B 0,C 180,E1 20430.896,E2 20430.896} C_VEL
LIN {X 0,Y 575.915,Z 1204.736,A -85,B 0,C 180,E1 20428.807,E2 20428.807} C_VEL
LIN {X 0,Y 575.913,Z 1203.51,A -85,B 0,C 180,E1 20426.417,E2 20426.417} C_VEL
LIN {X 0,Y 575.946,Z 1200.337,A -85,B 0,C 180,E1 20423.621,E2 20423.621} C_VEL
LIN {X 0,Y 576.025,Z 1195.923,A -85,B 0,C 180,E1 20421.113,E2 20421.113} C_VEL
LIN {X 0,Y 576.176,Z 1190.583,A -85,B 0,C 180,E1 20418.793,E2 20418.793} C_VEL
LIN {X 0,Y 576.568,Z 1182.685,A -85,B 0,C 180,E1 20416.052,E2 20416.052} C_VEL
LIN {X 0,Y 577.161,Z 1173.113,A -85,B 0,C 180,E1 20413.391,E2 20413.391} C_VEL
LIN {X 0,Y 577.893,Z 1164.073,A -85,B 0,C 180,E1 20411.228,E2 20411.228} C_VEL
LIN {X 0,Y 578.925,Z 1153.208,A -85,B 0,C 180,E1 20408.947,E2 20408.947} C_VEL
LIN {X 0,Y 580.563,Z 1138.275,A -85,B 0,C 180,E1 20406.234,E2 20406.234} C_VEL
LIN {X 0,Y 582.162,Z 1125.083,A -85,B 0,C 180,E1 20404.136,E2 20404.136} C_VEL
LIN {X 0,Y 584.064,Z 1111.07,A -85,B 0,C 180,E1 20402.138,E2 20402.138} C_VEL
LIN {X 0,Y 586.667,Z 1092.853,A -85,B 0,C 180,E1 20399.817,E2 20399.817} C_VEL
LIN {X 0,Y 589.385,Z 1074.491,A -85,B 0,C 180,E1 20397.776,E2 20397.776} C_VEL
LIN {X 0,Y 591.896,Z 1057.939,A -85,B 0,C 180,E1 20396.12,E2 20396.12} C_VEL
LIN {X 0,Y 594.593,Z 1040.391,A -85,B 0,C 180,E1 20394.539,E2 20394.539} C_VEL
LIN {X 0,Y 598.029,Z 1017.907,A -85,B 0,C 180,E1 20392.737,E2 20392.737} C_VEL
LIN {X 0,Y 601.143,Z 996.311,A -85,B 0,C 180,E1 20391.234,E2 20391.234} C_VEL
LIN {X 0,Y 603.894,Z 976.726,A -85,B 0,C 180,E1 20390.028,E2 20390.028} C_VEL
LIN {X 0,Y 606.434,Z 957.676,A -85,B 0,C 180,E1 20388.989,E2 20388.989} C_VEL
LIN {X 0,Y 608.833,Z 938.257,A -85,B 0,C 180,E1 20388.056,E2 20388.056} C_VEL
LIN {X 0,Y 611.339,Z 915.804,A -85,B 0,C 180,E1 20387.117,E2 20387.117} C_VEL
LIN {X 0,Y 614.037,Z 888.071,A -85,B 0,C 180,E1 20386.166,E2 20386.166} C_VEL
LIN {X 0,Y 615.873,Z 865.599,A -85,B 0,C 180,E1 20385.546,E2 20385.546} C_VEL
LIN {X 0,Y 617.3,Z 844.405,A -85,B 0,C 180,E1 20385.077,E2 20385.077} C_VEL
LIN {X 0,Y 618.449,Z 822.046,A -85,B 0,C 180,E1 20384.697,E2 20384.697} C_VEL
LIN {X 0,Y 624.378,Z 603.142,A -85,B 0,C 180,E1 20381.64,E2 20381.64} C_VEL
LIN {X 0,Y 629.778,Z 416.757,A -85,B 0,C 180,E1 20378.972,E2 20378.972} C_VEL
LIN {X 0,Y 616.899,Z 397.153,A -85,B 0,C 180,E1 20377.024,E2 20377.024} C_VEL
LIN {X 0,Y 607.319,Z 383.328,A -85,B 0,C 180,E1 20375.447,E2 20375.447} C_VEL
LIN {X 0,Y 599.982,Z 373.665,A -85,B 0,C 180,E1 20374.168,E2 20374.168} C_VEL
LIN {X 0,Y 595.675,Z 368.001,A -85,B 0,C 180,E1 20373.378,E2 20373.378} C_VEL
LIN {X 0,Y 591.576,Z 362.756,A -85,B 0,C 180,E1 20372.599,E2 20372.599} C_VEL
LIN {X 0,Y 586.153,Z 355.971,A -85,B 0,C 180,E1 20371.523,E2 20371.523} C_VEL
LIN {X 0,Y 583.131,Z 352.313,A -85,B 0,C 180,E1 20370.901,E2 20370.901} C_VEL
LIN {X 0,Y 580.412,Z 348.811,A -85,B 0,C 180,E1 20370.315,E2 20370.315} C_VEL
LIN {X 0,Y 579.863,Z 347.244,A -85,B 0,C 180,E1 20370.004,E2 20370.004} C_VEL
LIN {X 0,Y 577.761,Z 344.349,A -85,B 0,C 180,E1 20369.212,E2 20369.212} C_VEL
LIN {X 0,Y 577.246,Z 342.321,A -85,B 0,C 180,E1 20368.782,E2 20368.782} C_VEL
LIN {X 0,Y 577.229,Z 342.294,A -85,B 0,C 180,E1 20365.442,E2 20365.442} C_VEL
LIN {X 0,Y 577.242,Z 342.294,A -85,B 0,C 180,E1 20362.597,E2 20362.597} C_VEL
LIN {X 0,Y 577.225,Z 342.33,A -85,B 0,C 180,E1 20359.257,E2 20359.257} C_VEL
LIN {X 0,Y 577.262,Z 342.279,A -85,B 0,C 180,E1 20356.193,E2 20356.193} C_VEL
LIN {X 0,Y 577.22,Z 342.319,A -85,B 0,C 180,E1 20353.116,E2 20353.116} C_VEL
LIN {X 0,Y 577.263,Z 342.293,A -85,B 0,C 180,E1 20350.075,E2 20350.075} C_VEL
LIN {X 0,Y 577.224,Z 342.297,A -85,B 0,C 180,E1 20346.965,E2 20346.965} C_VEL
LIN {X 0,Y 577.266,Z 342.311,A -85,B 0,C 180,E1 20343.973,E2 20343.973} C_VEL
LIN {X 0,Y 577.227,Z 342.283,A -85,B 0,C 180,E1 20340.794,E2 20340.794} C_VEL
LIN {X 0,Y 577.263,Z 342.321,A -85,B 0,C 180,E1 20337.915,E2 20337.915} C_VEL
LIN {X 0,Y 577.23,Z 342.28,A -85,B 0,C 180,E1 20334.633,E2 20334.633} C_VEL
LIN {X 0,Y 577.274,Z 342.322,A -85,B 0,C 180,E1 20331.734,E2 20331.734} C_VEL
LIN {X 0,Y 577.241,Z 342.29,A -85,B 0,C 180,E1 20328.51,E2 20328.51} C_VEL
LIN {X 0,Y 577.286,Z 342.288,A -85,B 0,C 180,E1 20325.511,E2 20325.511} C_VEL
LIN {X 0,Y 577.249,Z 342.323,A -85,B 0,C 180,E1 20322.301,E2 20322.301} C_VEL
LIN {X 0,Y 577.309,Z 342.277,A -85,B 0,C 180,E1 20319.203,E2 20319.203} C_VEL
LIN {X 0,Y 577.283,Z 342.501,A -85,B 0,C 180,E1 20316.267,E2 20316.267} C_VEL
LIN {X 0,Y 578.559,Z 345.782,A -85,B 0,C 180,E1 20315.902,E2 20315.902} C_VEL
LIN {X 0,Y 581.225,Z 348.223,A -85,B 0,C 180,E1 20315.343,E2 20315.343} C_VEL
LIN {X 0,Y 582.497,Z 349.114,A -85,B 0,C 180,E1 20315.089,E2 20315.089} C_VEL
LIN {X 0,Y 584.687,Z 352.771,A -85,B 0,C 180,E1 20314.607,E2 20314.607} C_VEL
LIN {X 0,Y 587.807,Z 355.683,A -85,B 0,C 180,E1 20313.995,E2 20313.995} C_VEL
LIN {X 0,Y 590.758,Z 359.637,A -85,B 0,C 180,E1 20313.405,E2 20313.405} C_VEL
LIN {X 0,Y 593.251,Z 362.502,A -85,B 0,C 180,E1 20312.93,E2 20312.93} C_VEL
LIN {X 0,Y 600.755,Z 372.041,A -85,B 0,C 180,E1 20311.547,E2 20311.547} C_VEL
LIN {X 0,Y 608.553,Z 382.383,A -85,B 0,C 180,E1 20310.196,E2 20310.196} C_VEL
LIN {X 0,Y 617.383,Z 394.826,A -85,B 0,C 180,E1 20308.757,E2 20308.757} C_VEL
LIN {X 0,Y 629.761,Z 413.621,A -85,B 0,C 180,E1 20306.886,E2 20306.886} C_VEL
LIN {X 0,Y 623.192,Z 639.355,A -85,B 0,C 180,E1 20303.673,E2 20303.673} C_VEL
LIN {X 0,Y 621.162,Z 714.308,A -85,B 0,C 180,E1 20302.626,E2 20302.626} C_VEL
LIN {X 0,Y 620.289,Z 722.009,A -85,B 0,C 180,E1 20302.584,E2 20302.584} C_VEL
LIN {X 0,Y 615.417,Z 742.645,A -85,B 0,C 180,E1 20302.72,E2 20302.72} C_VEL
LIN {X 0,Y 614.71,Z 749.255,A -85,B 0,C 180,E1 20302.68,E2 20302.68} C_VEL
LIN {X 0,Y 612.562,Z 819.54,A -85,B 0,C 180,E1 20301.681,E2 20301.681} C_VEL
LIN {X 0,Y 610.827,Z 847.992,A -85,B 0,C 180,E1 20301.133,E2 20301.133} C_VEL
LIN {X 0,Y 608.74,Z 873.048,A -85,B 0,C 180,E1 20300.477,E2 20300.477} C_VEL
LIN {X 0,Y 606.725,Z 893.918,A -85,B 0,C 180,E1 20299.803,E2 20299.803} C_VEL
LIN {X 0,Y 604.326,Z 915.547,A -85,B 0,C 180,E1 20298.978,E2 20298.978} C_VEL
LIN {X 0,Y 601.311,Z 940.235,A -85,B 0,C 180,E1 20297.869,E2 20297.869} C_VEL
LIN {X 0,Y 597.847,Z 964.987,A -85,B 0,C 180,E1 20296.539,E2 20296.539} C_VEL
LIN {X 0,Y 594.906,Z 984.915,A -85,B 0,C 180,E1 20295.311,E2 20295.311} C_VEL
LIN {X 0,Y 591.924,Z 1004.314,A -85,B 0,C 180,E1 20293.968,E2 20293.968} C_VEL
LIN {X 0,Y 588.348,Z 1027.224,A -85,B 0,C 180,E1 20292.166,E2 20292.166} C_VEL
LIN {X 0,Y 585.091,Z 1047.167,A -85,B 0,C 180,E1 20290.366,E2 20290.366} C_VEL
LIN {X 0,Y 582.469,Z 1063.415,A -85,B 0,C 180,E1 20288.733,E2 20288.733} C_VEL
LIN {X 0,Y 579.908,Z 1079.624,A -85,B 0,C 180,E1 20286.928,E2 20286.928} C_VEL
LIN {X 0,Y 576.996,Z 1098.842,A -85,B 0,C 180,E1 20284.517,E2 20284.517} C_VEL
LIN {X 0,Y 574.841,Z 1113.703,A -85,B 0,C 180,E1 20282.393,E2 20282.393} C_VEL
LIN {X 0,Y 573.059,Z 1127.03,A -85,B 0,C 180,E1 20280.266,E2 20280.266} C_VEL
LIN {X 0,Y 571.38,Z 1141.329,A -85,B 0,C 180,E1 20277.689,E2 20277.689} C_VEL
LIN {X 0,Y 570.092,Z 1153.557,A -85,B 0,C 180,E1 20275.115,E2 20275.115} C_VEL
LIN {X 0,Y 569.277,Z 1162.963,A -85,B 0,C 180,E1 20272.84,E2 20272.84} C_VEL
LIN {X 0,Y 568.667,Z 1171.76,A -85,B 0,C 180,E1 20270.373,E2 20270.373} C_VEL
LIN {X 0,Y 568.253,Z 1179.852,A -85,B 0,C 180,E1 20267.616,E2 20267.616} C_VEL
LIN {X 0,Y 568.039,Z 1185.653,A -85,B 0,C 180,E1 20265.1,E2 20265.1} C_VEL
LIN {X 0,Y 567.949,Z 1189.882,A -85,B 0,C 180,E1 20262.712,E2 20262.712} C_VEL
LIN {X 0,Y 567.916,Z 1193.151,A -85,B 0,C 180,E1 20260.037,E2 20260.037} C_VEL
LIN {X 0,Y 567.912,Z 1194.664,A -85,B 0,C 180,E1 20257.486,E2 20257.486} C_VEL
LIN {X 0,Y 567.902,Z 1194.85,A -85,B 0,C 180,E1 20255.253,E2 20255.253} C_VEL
LIN {X 0,Y 567.911,Z 1193.984,A -85,B 0,C 180,E1 20253.027,E2 20253.027} C_VEL
LIN {X 0,Y 567.927,Z 1191.884,A -85,B 0,C 180,E1 20250.706,E2 20250.706} C_VEL
LIN {X 0,Y 567.979,Z 1188.285,A -85,B 0,C 180,E1 20248.184,E2 20248.184} C_VEL
LIN {X 0,Y 568.129,Z 1182.731,A -85,B 0,C 180,E1 20245.457,E2 20245.457} C_VEL
LIN {X 0,Y 568.431,Z 1176.031,A -85,B 0,C 180,E1 20242.927,E2 20242.927} C_VEL
LIN {X 0,Y 568.862,Z 1168.549,A -85,B 0,C 180,E1 20240.592,E2 20240.592} C_VEL
LIN {X 0,Y 569.662,Z 1158.561,A -85,B 0,C 180,E1 20237.944,E2 20237.944} C_VEL
LIN {X 0,Y 570.732,Z 1147.049,A -85,B 0,C 180,E1 20235.387,E2 20235.387} C_VEL
LIN {X 0,Y 571.945,Z 1136.034,A -85,B 0,C 180,E1 20233.234,E2 20233.234} C_VEL
LIN {X 0,Y 573.593,Z 1123.033,A -85,B 0,C 180,E1 20230.975,E2 20230.975} C_VEL
